ABB RobotStudio station: OpenRobotica_versão15_04_SEM_LETRAS_MASFUNC.rspag

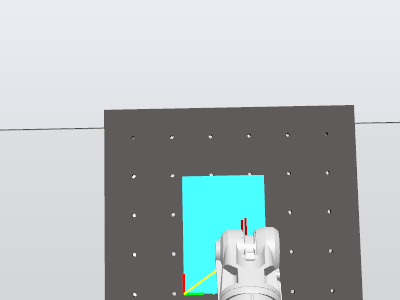
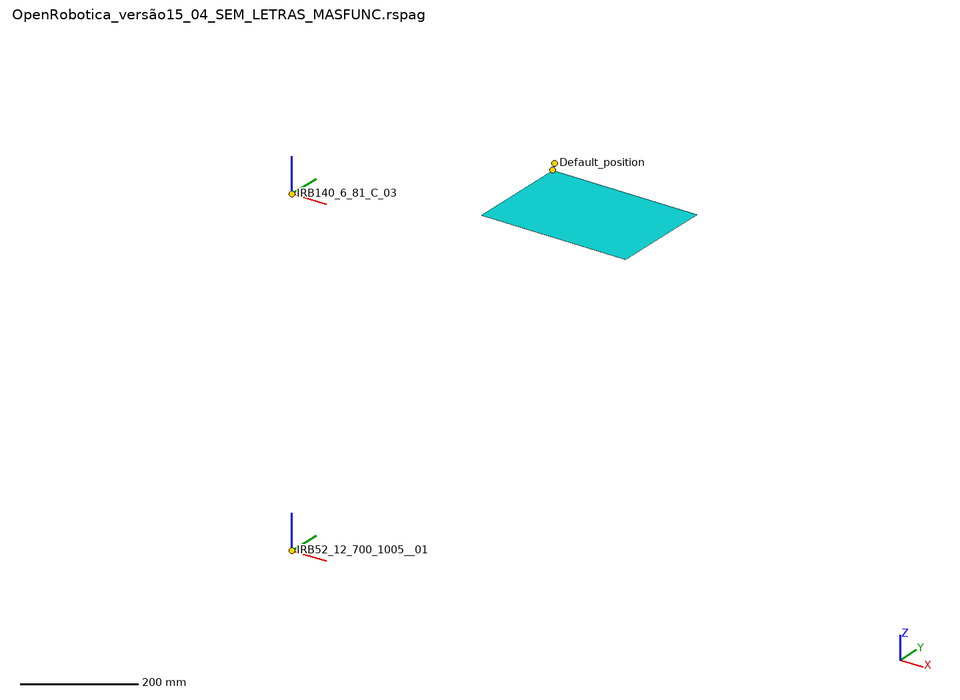
[picture v1: parts stored in the station drawn from their meshes, with robot base, taught points and paths (robot models come from the ABB library and are not in the file)]
--- station ---
Station V1 (saved by RobotStudio 24.1.10693.0)
Controller Robot_ISEP_IRB140, task T_ROB1: task frame (RAPID world) sits at (0, 0, 670) mm in the station
Controller Robot_ISEP_IRB140
  mechanical unit ROB_1: IRB140_6_81_C_03, 6 joints, base frame (0, 0, 0) mm
Controller Robo_open_v2
  mechanical unit ROB_1: IRB52_12_700_1005__01, 6 joints, base frame (0, 0, 0) mm, rotated rx 0 ry 0 rz 90 deg
Layout (positions relative to the parent item):
  - IRB140_6_81_C_03 [mechanism, from %ABB.RobotStudio.Models.IRB140%\IRB140_6_81_C_G_03.rslib] at (0, 0, 670) mm; joint values [-0.036, 0.5458, 0.1215, 0, 0.9034, 3.1056] (rad or m)
  - rob-table [part, from Libraries\rob-table.rslib]
  - pen [mechanism, from Libraries\pen.rslib] at (555, -20, 1029.5) mm, rotated rx 180 ry 0 rz 0 deg
  - paper [part, from Libraries\paper.rslib]
  - IRB52_12_700_1005__01 [mechanism, from %ABB.RobotStudio.Models.IRB52%\IRB52_12_700_1005_G_01.rslib] at (0, 0, 0) mm, rotated rx 0 ry 0 rz 90 deg; joint values [0, 0, 0, 0, 0, 0] (rad or m)
  - A3_Vertical [part] at (450, 125, 790) mm, rotated rx 0 ry 0 rz -90 deg, size 297 x 420 x 0.5 mm
  - A3_Horizontal [part] at (747, 125, 790) mm, rotated rx 0 ry 0 rz 180 deg, size 297 x 420 x 0.5 mm
  - A4_Vertical [part] at (450, 125, 790) mm, rotated rx 0 ry 0 rz -90 deg, size 210 x 297 x 0.5 mm
  - A4_Horizontal [part] at (450, -172, 790) mm, size 210 x 297 x 0.5 mm
  - A5_Vertical [part] at (450, 125, 790) mm, rotated rx 0 ry 0 rz -90 deg, size 148 x 210 x 0.5 mm
  - A5_Horizontal [part] at (450, -85, 790) mm, size 148 x 210 x 0.5 mm
Attachment: pen is attached to IRB140_6_81_C_03 / Link6
Targets, tools, work objects and paths stored in the station and not in the controller backup, written as RAPID:
! task T_ROB1
MODULE Module1
  CONST robtarget Target_Start:=[[0,0,0],[1,0,0,0],[0,0,0,0],[9E+09,9E+09,9E+09,9E+09,9E+09,9E+09]];
ENDMODULE

! task T_ROB1
MODULE DryLetter
  VAR robtarget up_inf_esq1:=[[0,0,0],[1,0,0,0],[0,0,0,0],[9E+09,9E+09,9E+09,9E+09,9E+09,9E+09]];
  VAR robtarget inf_esq1:=[[0,0,0],[1,0,0,0],[0,0,0,0],[9E+09,9E+09,9E+09,9E+09,9E+09,9E+09]];
  VAR robtarget sup_esq:=[[0,0,0],[1,0,0,0],[0,0,0,0],[9E+09,9E+09,9E+09,9E+09,9E+09,9E+09]];
  VAR robtarget sup_dir:=[[0,0,0],[1,0,0,0],[0,0,0,0],[9E+09,9E+09,9E+09,9E+09,9E+09,9E+09]];
  VAR robtarget inf_dir2:=[[0,0,0],[1,0,0,0],[0,0,0,0],[9E+09,9E+09,9E+09,9E+09,9E+09,9E+09]];
  VAR robtarget up_inf_dir2:=[[0,0,0],[1,0,0,0],[0,0,0,0],[9E+09,9E+09,9E+09,9E+09,9E+09,9E+09]];
  VAR robtarget meio_dir:=[[0,0,0],[1,0,0,0],[0,0,0,0],[9E+09,9E+09,9E+09,9E+09,9E+09,9E+09]];
  VAR robtarget meio_esq:=[[0,0,0],[1,0,0,0],[0,0,0,0],[9E+09,9E+09,9E+09,9E+09,9E+09,9E+09]];
  VAR robtarget up_final:=[[0,0,0],[1,0,0,0],[0,0,0,0],[9E+09,9E+09,9E+09,9E+09,9E+09,9E+09]];
  VAR robtarget sup_centro:=[[0,0,0],[1,0,0,0],[0,0,0,0],[9E+09,9E+09,9E+09,9E+09,9E+09,9E+09]];
  VAR robtarget meio_centro:=[[0,0,0],[1,0,0,0],[0,0,0,0],[9E+09,9E+09,9E+09,9E+09,9E+09,9E+09]];
  VAR robtarget inf_centro:=[[0,0,0],[1,0,0,0],[0,0,0,0],[9E+09,9E+09,9E+09,9E+09,9E+09,9E+09]];
  VAR robtarget up_meio_esq:=[[0,0,0],[1,0,0,0],[0,0,0,0],[9E+09,9E+09,9E+09,9E+09,9E+09,9E+09]];
  VAR robtarget sup_dir_meio:=[[0,0,0],[1,0,0,0],[0,0,0,0],[9E+09,9E+09,9E+09,9E+09,9E+09,9E+09]];
  VAR robtarget inf_dir_meio:=[[0,0,0],[1,0,0,0],[0,0,0,0],[9E+09,9E+09,9E+09,9E+09,9E+09,9E+09]];
  PROC Letra_A()
    MoveJ up_inf_esq1,v100,fine,pen\WObj:=Workobject_Paper;
    MoveL inf_esq1,v100,fine,pen\WObj:=Workobject_Paper;
    MoveL sup_esq,v100,z0,pen\WObj:=Workobject_Paper;
    MoveL sup_dir,v100,z0,pen\WObj:=Workobject_Paper;
    MoveL inf_dir2,v100,fine,pen\WObj:=Workobject_Paper;
    MoveL up_inf_dir2,v100,z0,pen\WObj:=Workobject_Paper;
    MoveL meio_dir,v100,z0,pen\WObj:=Workobject_Paper;
    MoveL meio_esq,v100,fine,pen\WObj:=Workobject_Paper;
    MoveL up_final,v100,z0,pen\WObj:=Workobject_Paper;
  ENDPROC
  PROC Letra_B()
    MoveJ target_oInf1Esq1,v100,fine,pen\WObj:=Workobject_Paper;
    MoveL target_oInf1Esq1,v100,fine,pen\WObj:=Workobject_Paper;
    MoveL target_oInf1Esq1,v100,fine,pen\WObj:=Workobject_Paper;
  ENDPROC
  PROC Letra_F()
    MoveJ up_inf_esq1,v100,fine,pen\WObj:=Workobject_Paper;
  ENDPROC
  PROC Space_letter()
    MoveJ target_oInf1Esq1,v100,fine,pen\WObj:=Workobject_Paper;
  ENDPROC
ENDMODULE

! task T_ROB1
MODULE Math
  PROC impressmenu()
    write_string;
    calculo_size;
    settingsTextMenu;
    settingsPageMenu;
    write_string;
    impress_mecanism;
  ENDPROC
ENDMODULE

! task T_ROB1
MODULE Menu
  PROC start_default()
    WaitTime 3;
  ENDPROC
  PROC principal_menu()
    menu_text;
    menu_paper;
    impressmenu;
  ENDPROC
ENDMODULE

! task T_ROB1
MODULE Print
  PROC impress_mecanism()
    draw;
    MoveJ Default_position,v1000,fine,pen\WObj:=Workobject_Paper;
    WaitTime 5;
  ENDPROC
ENDMODULE

! task T_ROB1
MODULE Fonts
  VAR robtarget target_oInf2Centro:=[[0,0,0],[1,0,0,0],[0,0,0,0],[9E+09,9E+09,9E+09,9E+09,9E+09,9E+09]];
  VAR robtarget target_oInf2Esq2:=[[0,0,0],[1,0,0,0],[0,0,0,0],[9E+09,9E+09,9E+09,9E+09,9E+09,9E+09]];
  VAR robtarget target_oInf2Dir1:=[[0,0,0],[1,0,0,0],[0,0,0,0],[9E+09,9E+09,9E+09,9E+09,9E+09,9E+09]];
  VAR robtarget target_oCentroDir1:=[[0,0,0],[1,0,0,0],[0,0,0,0],[9E+09,9E+09,9E+09,9E+09,9E+09,9E+09]];
  VAR robtarget target_oSup1Dir1:=[[0,0,0],[1,0,0,0],[0,0,0,0],[9E+09,9E+09,9E+09,9E+09,9E+09,9E+09]];
  VAR robtarget target_oSup2Esq2:=[[0,0,0],[1,0,0,0],[0,0,0,0],[9E+09,9E+09,9E+09,9E+09,9E+09,9E+09]];
  VAR robtarget target_oSup2Centro:=[[0,0,0],[1,0,0,0],[0,0,0,0],[9E+09,9E+09,9E+09,9E+09,9E+09,9E+09]];
  VAR robtarget target_oSup2Dir1:=[[0,0,0],[1,0,0,0],[0,0,0,0],[9E+09,9E+09,9E+09,9E+09,9E+09,9E+09]];
ENDMODULE


--- Backups/Robot_ISEP_IRB140/RAPID/TASK1/PROGMOD/CalibData.mod ---
MODULE CalibData
    PERS tooldata tWeldGun:=[TRUE,[[125.800591275,0,391.268161315],[0.898794046,0,0.438371147,0]],[3,[0,0,100],[0,1,0,0],0,0,0]];
    PERS tooldata pen:=[TRUE,[[0,0,139],[1,0,0,0]],[0.5,[0,0,20],[1,0,0,0],0,0,0]];
    TASK PERS wobjdata Workobject_Paper:=[FALSE,TRUE,"",[[450,125,118],[0,1,0,0]],[[50,50,0],[1,0,0,0]]];

    CONST robtarget Origem:=[[-50,-50,-2.5],[1,0,0,0],[0,0,0,0],[9E+09,9E+09,9E+09,9E+09,9E+09,9E+09]];
    CONST robtarget Default_position:=[[55,95,-102.5],[1,0,0,0],[0,0,0,0],[9E+09,9E+09,9E+09,9E+09,9E+09,9E+09]];
ENDMODULE

--- Backups/Robot_ISEP_IRB140/RAPID/TASK1/PROGMOD/Fonts.mod ---
MODULE Fonts

    ! Offset Z
    VAR num offsetZ := 10;

    ! On the paper

    VAR robtarget target_oInf1Esq1;
    VAR robtarget target_oInf1Esq2;
    VAR robtarget target_oInf1Centro;
    VAR robtarget target_oInf1Dir1;
    VAR robtarget target_oInf1Dir2;

    VAR robtarget target_oInf2Esq1;
    VAR robtarget target_oInf2Esq2;
    VAR robtarget target_oInf2Centro;
    VAR robtarget target_oInf2Dir1;
    VAR robtarget target_oInf2Dir2;

    VAR robtarget target_oCentroEsq1;
    VAR robtarget target_oCentroEsq2;
    VAR robtarget target_oCentroCentro;
    VAR robtarget target_oCentroDir1;
    VAR robtarget target_oCentroDir2;

    VAR robtarget target_oSup1Esq1;
    VAR robtarget target_oSup1Esq2;
    VAR robtarget target_oSup1Centro;
    VAR robtarget target_oSup1Dir1;
    VAR robtarget target_oSup1Dir2;

    VAR robtarget target_oSup2Esq1;
    VAR robtarget target_oSup2Esq2;
    VAR robtarget target_oSup2Centro;
    VAR robtarget target_oSup2Dir1;
    VAR robtarget target_oSup2Dir2;

    ! Above the paper

    VAR robtarget target_aInf1Esq1;
    VAR robtarget target_aInf1Esq2;
    VAR robtarget target_aInf1Centro;
    VAR robtarget target_aInf1Dir1;
    VAR robtarget target_aInf1Dir2;

    VAR robtarget target_aInf2Esq1;
    VAR robtarget target_aInf2Esq2;
    VAR robtarget target_aInf2Centro;
    VAR robtarget target_aInf2Dir1;
    VAR robtarget target_aInf2Dir2;

    VAR robtarget target_aCentroEsq1;
    VAR robtarget target_aCentroEsq2;
    VAR robtarget target_aCentroCentro;
    VAR robtarget target_aCentroDir1;
    VAR robtarget target_aCentroDir2;

    VAR robtarget target_aSup1Esq1;
    VAR robtarget target_aSup1Esq2;
    VAR robtarget target_aSup1Centro;
    VAR robtarget target_aSup1Dir1;
    VAR robtarget target_aSup1Dir2;

    VAR robtarget target_aSup2Esq1;
    VAR robtarget target_aSup2Esq2;
    VAR robtarget target_aSup2Centro;
    VAR robtarget target_aSup2Dir1;
    VAR robtarget target_aSup2Dir2;

    ! Last Position
    VAR robtarget last_position;

PROC draw( )

       TPWrite "Caracter a Imprimir: " + character;

       target_aInf1Esq1 := Offs(origem, coord_y_letter, coord_x_letter, -offsetZ);
       target_oInf1Esq1 := Offs(origem, coord_y_letter, coord_x_letter, 0);
       target_aInf1Dir2 := Offs(target_aInf1Esq1, 0, comprimento_letras,0);
       target_oInf1Dir2 := Offs(target_oInf1Esq1, 0, comprimento_letras,0);

       target_aSup1Esq1 := Offs(target_aInf1Esq1, altura_letras, 0, 0);
       target_oSup1Esq1 := Offs(target_oInf1Esq1, altura_letras, 0, 0);
       target_aSup1Dir2 := Offs(target_aSup1Esq1, 0, comprimento_letras,0);
       target_oSup1Dir2 := Offs(target_oSup1Esq1, 0, comprimento_letras,0);

       IF "Classic" = text_FontType THEN
	        IF "A" = character OR "a" = character THEN
	            ! Instructions to draw letter "A"
                    target_oCentroDir2 := Offs (target_oInf1Dir2, altura_letras/2 , 0, 0);
                    target_oCentroEsq1 := Offs (target_oCentroDir2, 0, -comprimento_letras, 0);
                    target_aCentroEsq1 := Offs (target_oCentroEsq1, 0, 0, -10);

                ! definição Trajeto

                    ! adaptar origem

                    MoveJ target_aInf1Esq1, v100, fine, pen\WObj:=Workobject_Paper;
                    MoveL target_oInf1Esq1, v100, fine, pen\WObj:=Workobject_Paper;
                    MoveL target_oSup1Esq1, v100, z50, pen\WObj:=Workobject_Paper;
                    MoveL target_oSup1Dir2, v100, z50, pen\WObj:=Workobject_Paper;
                    MoveL target_oInf1Dir2, v100, fine, pen\WObj:=Workobject_Paper;
                    MoveL target_oCentroDir2, v100, z0, pen\WObj:=Workobject_Paper;
                    MoveL target_oCentroEsq1, v100, fine, pen\WObj:=Workobject_Paper;
                    MoveL target_aCentroEsq1, v100, fine, pen\WObj:=Workobject_Paper;

                    !last_position := CRobT(\Tool:=pen\WObj:=Workobject_Paper);

	        ELSEIF "B" = character OR "b" = character THEN
	            ! Instructions to draw letter "B"
                target_oSup1Centro := Offs (target_oSup1Esq1, 0, comprimento_letras/2, 0);
                target_oSup2Dir2 := Offs (target_oSup1Centro, -altura_letras/4, comprimento_letras/2,0);
                target_oCentroCentro := Offs (target_oSup1Centro, -altura_letras/2, 0, 0); ! no MoveL tenho de fazer z30 (experimentar -> se quiser curva maior, fazer valor > 30)
                target_oInf2Dir2 := Offs (target_oCentroCentro, -altura_letras/4, comprimento_letras/2,0);
                target_oCentroEsq1 := Offs(target_oCentroCentro,0,-comprimento_letras/2, 0);
                target_oInf1Centro := Offs (target_oCentroCentro, -altura_letras/2, 0, 0); !z30

                ! definição Trajeto

                MoveJ target_oInf1Esq1, v100, fine, pen\WObj:=Workobject_Paper;
                MoveL target_oInf1Esq1, v100, fine, pen\WObj:=Workobject_Paper;
                MoveL target_oSup1Esq1, v100, fine, pen\WObj:=Workobject_Paper;
                MoveL target_oSup1Centro, v100, z0, pen\WObj:=Workobject_Paper;
                MoveC target_oSup2Dir2, target_oCentroCentro, v100, fine, pen\WObj:=Workobject_Paper;
                MoveL target_oCentroEsq1, v100, fine, pen\WObj:=Workobject_Paper;
                MoveL target_oCentroCentro, v100, fine, pen\WObj:=Workobject_Paper;
                MoveC target_oInf2Dir2 ,target_oInf1Centro, v100, fine, pen\WObj:=Workobject_Paper;
                MoveL target_oInf1Esq1, v100, fine, pen\WObj:=Workobject_Paper;

                MoveL target_aInf1Esq1, v100, z0, pen\WObj:=Workobject_Paper;

                last_position := CRobT(\Tool:=pen\WObj:=Workobject_Paper);

	        ELSEIF "C" = character OR "c" = character THEN
	            ! Instructions to draw letter "C"
                !Don't Finish

                target_oSup2Dir2 := Offs(target_oSup1Dir2,-altura_letras/4,0,0);
                target_aSup2Dir2 := Offs(target_oSup2Dir2,0,0, - offsetZ);
                target_oSup1Centro := Offs(target_oSup1Esq1,0,comprimento_letras/2,0);
                target_oSup2Esq1 := Offs(target_oSup1Esq1,-altura_letras/4,0,0);
                target_oInf2Esq1 := Offs(target_oInf1Esq1,altura_letras/4,0,0);
                target_oInf1Centro := Offs(target_oInf1Esq1,0,comprimento_letras/2,0);
                target_oInf2Dir2 := Offs(target_oInf1Esq1,altura_letras/4,0,0);
                target_aInf2Dir2 := Offs(target_oInf2Dir2,0,0, - offsetZ);


                !traject
                MoveJ target_aSup2Dir2, v100, fine, pen\WObj:=Workobject_Paper;
                MoveL target_oSup2Dir2, v100, fine, pen\WObj:=Workobject_Paper;
                MoveC target_oSup1Centro, target_oSup2Esq1, v100, fine, pen\WObj:=Workobject_Paper;
                MoveL target_oInf2Esq1, v100, fine, pen\WObj:=Workobject_Paper;
                MoveC target_oInf1Centro, target_oInf2Dir2, v100, fine, pen\WObj:=Workobject_Paper;
                MoveL target_aInf2Dir2, v100, fine, pen\WObj:=Workobject_Paper;

	        ELSEIF "D" = character OR "d" = character THEN
	            ! Instructions to draw letter "D"
	        ELSEIF "E" = character OR "e" = character THEN
	            ! Instructions to draw letter "E"
	        ELSEIF "F" = character OR "f" = character THEN
	            ! Instructions to draw letter "F"
	        ELSEIF "G" = character OR "g" = character THEN
	            ! Instructions to draw letter "G"
	        ELSEIF "H" = character OR "h" = character THEN
	            ! Instructions to draw letter "H"
	        ELSEIF "I" = character OR "i" = character THEN
	            ! Instructions to draw letter "I"
	        ELSEIF "J" = character OR "j" = character THEN
	            ! Instructions to draw letter "J"
	        ELSEIF "K" = character OR "k" = character THEN
	            ! Instructions to draw letter "K"
	        ELSEIF "L" = character OR "l" = character THEN
	            ! Instructions to draw letter "L"
	       ELSEIF "M" = character OR "m" = character THEN
	            ! Instructions to draw letter "M"
                target_aCentroCentro := Offs( target_aInf1Esq1 , altura_letras/2 , comprimento_letras/2 , 0);
                target_oCentroCentro := Offs( target_oInf1Esq1 , altura_letras/2 , comprimento_letras/2 , 0);

		        ! Movement
		        MoveJ target_aInf1Esq1, v100, fine, pen\WObj:=Workobject_Paper;
		        MoveL target_oInf1Esq1, v100, fine, pen\WObj:=Workobject_Paper;
		        MoveL target_oSup1Esq1, v100, fine, pen\WObj:=Workobject_Paper;
		        MoveL target_oCentroCentro, v100, fine, pen\WObj:=Workobject_Paper;
		        MoveL target_oSup1Dir2, v100, fine, pen\WObj:=Workobject_Paper;
		        MoveL target_oInf1Dir2, v100, fine, pen\WObj:=Workobject_Paper;
		        MoveL target_aInf1Dir2, v100, fine, pen\WObj:=Workobject_Paper;

	        ELSEIF "N" = character OR "n" = character THEN
		        ! Movement
		        MoveJ target_aInf1Esq1, v100, fine, pen\WObj:=Workobject_Paper;
		        MoveL target_oInf1Esq1, v100, fine, pen\WObj:=Workobject_Paper;
		        MoveL target_oSup1Esq1, v100, fine, pen\WObj:=Workobject_Paper;
		        MoveL target_oInf1Dir2, v100, fine, pen\WObj:=Workobject_Paper;
		        MoveL target_oSup1Dir2, v100, fine, pen\WObj:=Workobject_Paper;
		        MoveL target_aSup1Dir2, v100, fine, pen\WObj:=Workobject_Paper;

	        ELSEIF "O" = character OR "o" = character THEN
	            ! Instructions to draw letter "O"
                target_aSup1Centro := Offs( target_aInf1Esq1 , altura_letras , comprimento_letras/2 , 0);
                target_oSup1Centro := Offs( target_oInf1Esq1 , altura_letras , comprimento_letras/2 , 0);

                target_aInf1Centro := Offs( target_aInf1Esq1 , 0 , comprimento_letras/2 , 0);
                target_oInf1Centro := Offs( target_oInf1Esq1 , 0 , comprimento_letras/2 , 0);

                target_aCentroDir2 := Offs( target_aInf1Esq1 , altura_letras/2 , comprimento_letras , 0);
                target_oCentroDir2 := Offs( target_oInf1Esq1 , altura_letras/2 , comprimento_letras , 0);

                target_aCentroEsq1 := Offs( target_aInf1Esq1 , altura_letras/2 , 0 , 0);
                target_oCentroEsq1 := Offs( target_oInf1Esq1 , altura_letras/2 , 0 , 0);


		        ! Movement
		        MoveJ target_aCentroEsq1, v100, fine, pen\WObj:=Workobject_Paper;
		        MoveL target_oCentroEsq1, v100, fine, pen\WObj:=Workobject_Paper;
		        MoveC target_oSup1Centro , target_oCentroDir2 , v100, fine, pen\WObj:=Workobject_Paper;
		        MoveC target_oInf1Centro , target_oCentroEsq1 , v100, fine, pen\WObj:=Workobject_Paper;
		        MoveL target_aCentroEsq1, v100, fine, pen\WObj:=Workobject_Paper;

	        ELSEIF "P" = character OR "p" = character THEN
	            ! Instructions to draw letter "P"
                target_aSup2Dir2 := Offs( target_aInf1Esq1 , altura_letras*3/4 , comprimento_letras, 0);
                target_oSup2Dir2 := Offs( target_oInf1Esq1 , altura_letras*3/4 , comprimento_letras, 0);

                target_aCentroEsq1 := Offs( target_aInf1Esq1 , altura_letras/2 , 0, 0);
                target_oCentroEsq1 := Offs( target_oInf1Esq1 , altura_letras/2 , 0, 0);

                target_aCentroEsq2 := Offs( target_aInf1Esq1 , altura_letras/2 , comprimento_letras *1/4, 0);
                target_oCentroEsq2 := Offs( target_oInf1Esq1 , altura_letras/2 , comprimento_letras *1/4, 0);

                target_aSup1Esq2 := Offs( target_aInf1Esq1 , altura_letras , comprimento_letras *1/4, 0);
                target_oSup1Esq2 := Offs( target_oInf1Esq1 , altura_letras , comprimento_letras *1/4, 0);

		        ! Movement
		        MoveJ target_aInf1Esq1, v100, fine, pen\WObj:=Workobject_Paper;
		        MoveL target_oInf1Esq1, v100, fine, pen\WObj:=Workobject_Paper;
		        MoveL target_oSup1Esq1, v100, fine, pen\WObj:=Workobject_Paper;
		        MoveL target_oSup1Esq2, v100, fine, pen\WObj:=Workobject_Paper;
		        MoveC target_oSup2Dir2 , target_oCentroEsq2 , v100, fine, pen\WObj:=Workobject_Paper;
		        MoveL target_oCentroEsq1, v100, fine, pen\WObj:=Workobject_Paper;
		        MoveL target_aCentroEsq1, v100, fine, pen\WObj:=Workobject_Paper;


	        ELSEIF "Q" = character OR "q" = character THEN
	            ! Instructions to draw letter "Q"
	        ELSEIF "R" = character OR "r" = character THEN
	            ! Instructions to draw letter "R"
	        ELSEIF "S" = character OR "s" = character THEN
	            ! Instructions to draw letter "S"
                target_aSup2Dir2 := Offs( target_aInf1Esq1 , altura_letras * 3/4 , comprimento_letras , 0);
                target_oSup2Dir2 := Offs( target_oInf1Esq1 , altura_letras * 3/4 , comprimento_letras , 0);


                target_aInf2Esq1 := Offs( target_aInf1Esq1 , altura_letras * 1/4 , 0 , 0);
                target_oInf2Esq1 := Offs( target_oInf1Esq1 , altura_letras * 1/4 , 0 , 0);

                target_aInf1Centro := Offs( target_aInf1Esq1 , 0 , comprimento_letras/2 , 0);
                target_oInf1Centro := Offs( target_oInf1Esq1 , 0 , comprimento_letras/2 , 0);
                target_aSup1Centro := Offs( target_aInf1Esq1 , altura_letras , comprimento_letras/2 , 0);
                target_oSup1Centro := Offs( target_oInf1Esq1 , altura_letras , comprimento_letras/2 , 0);

                target_aInf2Dir2 := Offs( target_aInf1Esq1 , altura_letras * 1/4 , comprimento_letras , 0);
                target_oInf2Dir2 := Offs( target_oInf1Esq1 , altura_letras * 1/4 , comprimento_letras , 0);

                target_aCentroCentro := Offs( target_aInf1Esq1 , altura_letras/2 , comprimento_letras/2 , 0);
                target_oCentroCentro := Offs( target_oInf1Esq1 , altura_letras/2 , comprimento_letras/2 , 0);

                target_aSup2Esq1 := Offs( target_aInf1Esq1 , altura_letras * 3/4 , 0 , 0);
                target_oSup2Esq1 := Offs( target_oInf1Esq1 , altura_letras * 3/4 , 0 , 0);

                target_oCentroEsq1 := Offs( target_oInf1Esq1, altura_letras / 2 ,0,0);

                target_oCentroDir2 := Offs ( target_oInf1Dir2, altura_letras / 2 , 0 , 0);
		        ! Movement
		        MoveJ target_aSup2Dir2, v100, fine, pen\WObj:=Workobject_Paper;
		        MoveL target_oSup2Dir2, v100, fine, pen\WObj:=Workobject_Paper;
		        MoveC target_oSup1Centro , target_oSup2Esq1 , v100, fine, pen\WObj:=Workobject_Paper;

                MoveL target_oCentroEsq1, v100, z150, pen\WObj:=Workobject_Paper;
                MoveL target_oCentroCentro, v100, fine, pen\WObj:=Workobject_Paper;
                MoveL target_oCentroDir2, v100, z150, pen\WObj:=Workobject_Paper;
                MoveL target_oInf2Dir2, v100, fine, pen\WObj:=Workobject_Paper;

                MoveC target_oInf1Centro , target_oInf2Esq1 , v100, fine, pen\WObj:=Workobject_Paper;
		        MoveL target_aInf2Esq1, v100, fine, pen\WObj:=Workobject_Paper;


	        ELSEIF "T" = character OR "t" = character THEN
	            ! Instructions to draw letter "T"
                target_aInf1Centro := Offs( target_aInf1Esq1 , 0 , comprimento_letras/2 , 0);
                target_oInf1Centro := Offs( target_oInf1Esq1 , 0 , comprimento_letras/2 , 0);
                target_aSup1Centro := Offs( target_aInf1Esq1 , altura_letras , comprimento_letras/2 , 0);
                target_oSup1Centro := Offs( target_oInf1Esq1 , altura_letras , comprimento_letras/2 , 0);

		        ! Movement
		        MoveJ target_aSup1Esq1, v100, fine, pen\WObj:=Workobject_Paper;
		        MoveL target_oSup1Esq1, v100, fine, pen\WObj:=Workobject_Paper;
		        MoveL target_oSup1Dir2, v100, fine, pen\WObj:=Workobject_Paper;
		        MoveL target_oSup1Centro, v100, fine, pen\WObj:=Workobject_Paper;
		        MoveL target_oInf1Centro, v100, fine, pen\WObj:=Workobject_Paper;
		        MoveL target_aInf1Centro, v100, fine, pen\WObj:=Workobject_Paper;

	        ELSEIF "U" = character OR "u" = character THEN
	            ! Instructions to draw letter "U"
                target_aInf1Centro := Offs( target_aInf1Esq1 , 0 , comprimento_letras/2 , 0);
                target_oInf1Centro := Offs( target_oInf1Esq1 , 0 , comprimento_letras/2 , 0);
                target_aInf2Esq1 := Offs( target_aInf1Esq1 , altura_letras/4 , 0 , 0);
                target_oInf2Esq1 := Offs( target_oInf1Esq1 , altura_letras/4 , 0 , 0);
                target_aInf2Dir2 := Offs( target_aInf1Esq1 , altura_letras/4 , comprimento_letras , 0);
                target_oInf2Dir2 := Offs( target_oInf1Esq1 , altura_letras/4 , comprimento_letras , 0);

		        ! Movement
		        MoveJ target_aSup1Esq1, v100, fine, pen\WObj:=Workobject_Paper;
		        MoveL target_oSup1Esq1, v100, fine, pen\WObj:=Workobject_Paper;
		        MoveL target_oInf2Esq1, v100, fine, pen\WObj:=Workobject_Paper;
		        MoveC target_oInf1Centro , target_oInf2Dir2 , v100, fine, pen\WObj:=Workobject_Paper;
		        MoveL target_oSup1Dir2, v100, fine, pen\WObj:=Workobject_Paper;
		        MoveL target_aSup1Dir2, v100, fine, pen\WObj:=Workobject_Paper;


	        ELSEIF "V" = character OR "v" = character THEN
	            ! Instructions to draw letter "V"
                target_aInf1Centro := Offs( target_aInf1Esq1 , 0 , comprimento_letras/2 , 0);
                target_oInf1Centro := Offs( target_oInf1Esq1 , 0 , comprimento_letras/2 , 0);

		        ! Movement
		        MoveJ target_aSup1Esq1, v100, fine, pen\WObj:=Workobject_Paper;
		        MoveL target_oSup1Esq1, v100, fine, pen\WObj:=Workobject_Paper;
		        MoveL target_oInf1Centro, v100, fine, pen\WObj:=Workobject_Paper;
		        MoveL target_oSup1Dir2, v100, fine, pen\WObj:=Workobject_Paper;
		        MoveL target_aSup1Dir2, v100, fine, pen\WObj:=Workobject_Paper;
		        !MoveL target_aInf1Dir2, v100, fine, pen\WObj:=Workobject_Paper;

	        ELSEIF "W" = character OR "w" = character THEN
	            ! Instructions to draw letter "W"
                target_aCentroCentro := Offs( target_aInf1Esq1 , altura_letras/2 , comprimento_letras/2 , 0);
                target_oCentroCentro := Offs( target_oInf1Esq1 , altura_letras/2 , comprimento_letras/2 , 0);
                target_aInf1Esq2 := Offs( target_aInf1Esq1 , 0 , comprimento_letras/4 , 0);
                target_oInf1Esq2 := Offs( target_oInf1Esq1 , 0 , comprimento_letras/4 , 0);
                target_aInf1Dir1 := Offs( target_aInf1Esq1 , 0 , comprimento_letras*3/4 , 0);
                target_oInf1Dir1 := Offs( target_oInf1Esq1 , 0 , comprimento_letras*3/4 , 0);

		        ! Movement
		        MoveJ target_aSup1Esq1, v100, fine, pen\WObj:=Workobject_Paper;
		        MoveL target_oSup1Esq1, v100, fine, pen\WObj:=Workobject_Paper;
		        MoveL target_oInf1Esq2, v100, fine, pen\WObj:=Workobject_Paper;
		        MoveL target_oCentroCentro, v100, fine, pen\WObj:=Workobject_Paper;
		        MoveL target_oInf1Dir1, v100, fine, pen\WObj:=Workobject_Paper;
		        MoveL target_oSup1Dir2, v100, fine, pen\WObj:=Workobject_Paper;
		        MoveL target_aSup1Dir2, v100, fine, pen\WObj:=Workobject_Paper;
		        !MoveL target_aInf1Dir2, v100, fine, pen\WObj:=Workobject_Paper;

	        ELSEIF "X" = character OR "x" = character THEN
	            ! Instructions to draw letter "X"

		        ! Movement
		        MoveJ target_aSup1Esq1, v100, fine, pen\WObj:=Workobject_Paper;
		        MoveL target_oSup1Esq1, v100, fine, pen\WObj:=Workobject_Paper;
		        MoveL target_oInf1Dir2, v100, fine, pen\WObj:=Workobject_Paper;
		        MoveL target_aInf1Dir2, v100, fine, pen\WObj:=Workobject_Paper;
		        MoveL target_aSup1Dir2, v100, fine, pen\WObj:=Workobject_Paper;
		        MoveL target_oSup1Dir2, v100, fine, pen\WObj:=Workobject_Paper;
		        MoveL target_oInf1Esq1, v100, fine, pen\WObj:=Workobject_Paper;
		        MoveL target_aInf1Esq1, v100, fine, pen\WObj:=Workobject_Paper;
		        !MoveL target_aInf1Dir2, v100, fine, pen\WObj:=Workobject_Paper;

	        ELSEIF "Y" = character OR "y" = character THEN

	            ! Instructions to draw letter "Y"
                target_aCentroCentro := Offs( target_aInf1Esq1 , altura_letras/2 , comprimento_letras/2 , 0);
                target_oCentroCentro := Offs( target_oInf1Esq1 , altura_letras/2 , comprimento_letras/2 , 0);
                target_aInf1Centro := Offs( target_aInf1Esq1 , 0 , comprimento_letras/2 , 0);
                target_oInf1Centro := Offs( target_oInf1Esq1 , 0 , comprimento_letras/2 , 0);

		        ! Movement
		        MoveJ target_aSup1Esq1, v100, fine, pen\WObj:=Workobject_Paper;
		        MoveL target_oSup1Esq1, v100, fine, pen\WObj:=Workobject_Paper;
		        MoveL target_oCentroCentro, v100, fine, pen\WObj:=Workobject_Paper;
		        MoveL target_oSup1Dir2, v100, fine, pen\WObj:=Workobject_Paper;
		        MoveL target_aSup1Dir2, v100, fine, pen\WObj:=Workobject_Paper;
		        MoveL target_aCentroCentro, v100, fine, pen\WObj:=Workobject_Paper;
		        MoveL target_oCentroCentro, v100, fine, pen\WObj:=Workobject_Paper;
		        MoveL target_oInf1Centro, v100, fine, pen\WObj:=Workobject_Paper;
		        MoveL target_aInf1Centro, v100, fine, pen\WObj:=Workobject_Paper;
		        !MoveL target_aInf1Dir2, v100, fine, pen\WObj:=Workobject_Paper;

	        ELSEIF "Z" = character OR "z" = character THEN
	           ! Instructions to draw letter "Z"

		        ! Movement
		        MoveJ target_aSup1Esq1, v100, fine, pen\WObj:=Workobject_Paper;
		        MoveL target_oSup1Esq1, v100, fine, pen\WObj:=Workobject_Paper;
		        MoveL target_oSup1Dir2, v100, fine, pen\WObj:=Workobject_Paper;
		        MoveL target_oInf1Esq1, v100, fine, pen\WObj:=Workobject_Paper;
		        MoveL target_oInf1Dir2, v100, fine, pen\WObj:=Workobject_Paper;
		        MoveL target_aInf1Dir2, v100, fine, pen\WObj:=Workobject_Paper;

	        ELSEIF " " = character THEN
	            ! Instructions to draw letter " "
                MoveJ target_oInf1Esq1, v100, fine, pen\WObj:=Workobject_Paper;
	        ELSE

	        ENDIF
	      ENDIF
    ENDPROC
ENDMODULE

--- Backups/Robot_ISEP_IRB140/RAPID/TASK1/PROGMOD/MainModule.mod ---
MODULE MainModule

        CONST robtarget Target_10:=[[0,0,0],[1,0,0,0],[0,-1,-2,0],[9E+09,9E+09,9E+09,9E+09,9E+09,9E+09]];
    CONST robtarget Target_20:=[[70,30,0],[1,0,0,0],[0,-1,-2,0],[9E+09,9E+09,9E+09,9E+09,9E+09,9E+09]];
    CONST robtarget Target_30:=[[0,60,0],[1,0,0,0],[0,-1,-2,0],[9E+09,9E+09,9E+09,9E+09,9E+09,9E+09]];
PROC main()
       ! Default sequence to reposition the robot
       startDefault;

       ! Main loop
        WHILE TRUE DO
            mainMenu;
        ENDWHILE


    ENDPROC
    PROC Path_A()
    ENDPROC
ENDMODULE

--- Backups/Robot_ISEP_IRB140/RAPID/TASK1/PROGMOD/Math.mod ---
MODULE Math
    ! ============== Declara??o de Variaveis =======================

    ! Apoio para as perguntas
    VAR num answer_impress;

    ! Write array
    PERS string char_impress;

    VAR num userInputTextLenght := 0;
    VAR num workSpaceWidth;
    VAR num workSpaceLength;
    VAR num letterLenghtAutomated;
    VAR num letterWidthAutomated;
    VAR num text_SpaceLettersAutomated;

    CONST num factorSpaceBetweenLetters := 5;
    CONST num factorHightLetter := 2;

    ! Position text
    VAR num xAvailable := 0 ;
    VAR num yAvailable := 0 ;
    VAR num coord_x_letter;
    VAR num coord_y_letter;

    PROC write_string()
        TPWrite "Insira a(s) palavra(s) pretendida(s) para imprimir.";
        userInputText := UIAlphaEntry(
            \Header:= "Impressão",
            \Message:= ""
            \Icon:=iconInfo
            \InitString:= "OPEN ROBOTICA");
    ENDPROC


    PROC calculateSizeLetterAutomated()
        ! Get the amount of chars in the array of text
        userInputTextLenght := StrLen(userInputText);

        ! Garentee the user actually inserts a text
        IF 0 = userInputTextLenght THEN
              TPWrite "Error : Necessário texto para poder imprimir.";
              errorA := TRUE;
              RETURN ;
        ENDIF

        ! Get the size of the page
        workSpaceWidth := paper_Width - paper_LeftMargin - paper_RightMargin ;
        workSpaceLength := paper_Length - paper_TopMargin - paper_BottomMargin ;

        ! Calculate the width of the text acordingly to fit the page line
        letterWidthAutomated := ( workSpaceWidth - ( ( userInputTextLenght - 1 ) * text_SpaceLetters ) ) DIV userInputTextLenght ;

        FOR I FROM 1 TO 10 DO
            ! Calculate the space required between letters
            text_SpaceLettersAutomated := text_SpaceLetters + letterWidthAutomated DIV factorSpaceBetweenLetters ;

            ! Recalculate the lenght of the text acordingly to fit the page line considering the new spacement
            letterWidthAutomated := ( workSpaceWidth - ( ( userInputTextLenght - 1 ) * text_SpaceLettersAutomated ) ) DIV userInputTextLenght ;
        ENDFOR

        ! Garantee a minimum space between
        IF 0 = text_SpaceLettersAutomated THEN
             text_SpaceLettersAutomated := 0.1;
        ENDIF

        ! Calcule the necessary height of letter
        letterLenghtAutomated := letterWidthAutomated * factorHightLetter;

        IF workSpaceLength  < letterLenghtAutomated  THEN
            letterLenghtAutomated := workSpaceLength ;
        ENDIF
    ENDPROC

    PROC calculateOrigin( )
        IF FALSE = automatic THEN
	        IF "Esquerda" = paper_alignment THEN
	        	xAvailable := paper_LeftMargin;
	        ELSEIF "Direita" = paper_alignment THEN
	        	xAvailable := paper_RightMargin - letterWidthAutomated * userInputTextLenght ;
	        ELSEIF "Centrado" = paper_alignment THEN
	            xAvailable := workSpaceWidth / 2 - letterWidthAutomated * userInputTextLenght ;
	        ELSEIF "Justificado" = paper_alignment THEN
	        	xAvailable := paper_LeftMargin;
	        ENDIF
        ELSEIF TRUE = automatic THEN
	       	xAvailable := paper_LeftMargin;
	        IF 0 = yAvailable THEN
	            yAvailable := paper_Length - paper_TopMargin - letterLenghtAutomated;
	        ELSE
	            yAvailable := coord_y_letter - letterLenghtAutomated - text_SpaceParag ;
	            !Condition to out page
	            IF 0 > yAvailable THEN
                     TPWrite "Error : Fora de página";
                     errorA := TRUE;
                     RETURN;
	            ENDIF
	        ENDIF
        ENDIF

        coord_x_letter := xAvailable;
        coord_y_letter := yAvailable;
    ENDPROC
ENDMODULE

--- Backups/Robot_ISEP_IRB140/RAPID/TASK1/PROGMOD/Menu.mod ---
MODULE Menu

    ! ============== Definition of variables/constants =============================== !

    ! Questions suport
    VAR num answerInitMenu;
    VAR num answerPaperMenu;
    VAR num answerPaperMenu2;
    VAR num answerSettingMenu;
    VAR num answerWriteTextMenu;
    VAR num answerWriteTextMenu2;
    VAR num answerWrittingMenu;
    VAR num answerPrintingMenu;
    VAR num answerDebugMenu;

    ! Variable that stores the text input
    VAR string userInputText ;
    VAR string character;

    ! Dimensions of the format papers (mm)
    CONST num a3Lenght := 297;
    CONST num a3Width := 420;
    CONST num a4Lenght := 210;
    CONST num a4Width := 297;
    CONST num a5Lenght := 148;
    CONST num a5Width := 210;

    ! Initialize the paper characteristics
    VAR string paper_size := "A4";
    VAR string paper_orientation := "Vertical";
    VAR string paper_alignment := "Esquerda";
    VAR num paper_TopMargin := 20;
    VAR num paper_BottomMargin := 20;
    VAR num paper_LeftMargin := 10;
    VAR num paper_RightMargin := 10;
    VAR num paper_Width := a4Lenght;
    VAR num paper_Length := a4Width;

    ! Initialize the text characteristics
    VAR string text_FontType := "Classic";
    VAR num text_SizePT := 12;
    VAR string text_Color := "Black";
    VAR num text_Rotation := 0;
    VAR num text_SpaceLetters := 2;
    VAR num text_SpaceParag := 5;

    ! Initialize letters characteristics
    VAR num letter_lenght := 5;
    VAR num letter_width := 10;

    VAR num paragraph_write := 0;

    VAR bool automatic := FALSE;

    VAR num altura_letras;
    VAR num comprimento_letras;

    VAR bool errorA := FALSE;

    ! ==================== Code - default ========================= !

    ! Process for the inicialization program
    PROC startDefault( )
        ! Clear console
        TPErase;

        MoveJ Default_position,v1000,fine,pen\WObj:=Workobject_Paper;

        ! JumpHome; !TODO
        TPWrite "O robot está pronto a ser operado.";

        WaitTime(1);
    ENDPROC

    ! ==================== Code - mainMenu ======================== !

    PROC mainMenu()
        !Clear console
        TPErase;

        ! Welcome page.
        TPWrite "Plotter & Open Robótica";

        ! Options of the menu
        TPReadFK answerInitMenu ,
                 stEmpty ,
                 "Escrever Manualmente" ,
                 "Definições texto" ,
                 "Definições folha" ,
                 "Imprimir",
                 "Debug";

        IF 1 = answerInitMenu THEN
            writeTextMenu;
        ELSEIF 2 = answerInitMenu THEN
           answersettingMenu := 0;
           settingsTextMenu ;
        ELSEIF 3 = answerInitMenu THEN
            settingsPageMenu ;
        ELSEIF 4 = answerInitMenu THEN
            printingPageMenu ;
        ELSEIF 5 = answerInitMenu THEN
            debugMenu ;
        ENDIF
    ENDPROC

    ! ==================== Code - writeMenu ======================= !

    PROC writeTextMenu( )
        WHILE answerWrittingMenu <> 5 DO
            ! Clear the console
            TPErase;

            TPWrite("Frase a escrever:");
            ! Options to change settings of the page
            TPReadFK answerSettingMenu,
                     userInputText ,
                     "Escrever",
                     stEmpty,
                     stEmpty,
                     stEmpty,
                     "Voltar";

            IF 1 = answersettingMenu THEN
                write_string;

            ELSEIF 2 = answersettingMenu THEN

            ELSEIF 3 = answersettingMenu THEN

            ELSEIF 4 = answersettingMenu THEN

            ELSEIF 5 = answersettingMenu THEN
                answerWrittingMenu := 5;
                ! Back to menu
            ENDIF
        ENDWHILE
        answerWrittingMenu := 0;
    ENDPROC

    ! ==================== Code - settingsText ==================== !

    PROC settingsTextMenu( )
        WHILE answersettingMenu <> 5 DO
            ! Clear the console
            TPErase;

            tpWriteReportSettingsTextMenu;

            ! Options to change settings of the page
            TPReadFK answerSettingMenu,
                     stEmpty ,
                     "Fonte",
                     "Tamanho (pt)",
                     "Cor",
                     "Página seguinte",
                     "Voltar";

            IF 1 = answersettingMenu THEN
                fontTypePageMenu ;

            ELSEIF 2 = answersettingMenu THEN
                TPReadNum text_SizePT, "Qual é o tamanho da letra? (pt) (default = 12)";
                !TODO convert pt to mm

            ELSEIF 3 = answersettingMenu THEN
                fontColorPageMenu ;

            ELSEIF 4 = answersettingMenu THEN
                answersettingMenu := 0;
                settingsTextMenu2 ;

            ELSEIF 5 = answersettingMenu THEN
                answersettingMenu := 5;
                ! Back to menu
            ENDIF

        ENDWHILE
    ENDPROC

    PROC settingsTextMenu2( )
        WHILE answersettingMenu <> 5 DO
            ! Clear the console
            TPErase;

            tpWriteReportSettingsTextMenu;

            ! Options to change settings of the page
            TPReadFK answerSettingMenu,
                     stEmpty ,
                     "Rotação",
                     "Espaçamento entre letras",
                     "Espaçamento entre paragráfos",
                     "Página seguinte",
                     "Voltar";

            IF 1 = answersettingMenu THEN
                TPReadNum text_Rotation, "Qual é a rotação pretendida? (graus)";

            ELSEIF 2 = answersettingMenu THEN
                TPReadNum text_SpaceLetters, "Qual é o espaçamento entre letras? (mm) (default = 2)";

            ELSEIF 3 = answersettingMenu THEN
                TPReadNum text_SpaceParag, "Qual é o espaçamento entre paragráfos? (mm) (default = 5)";

            ELSEIF 4 = answersettingMenu THEN
                answersettingMenu := 0;
                settingsTextMenu3 ;

            ELSEIF 5 = answersettingMenu THEN
                answersettingMenu := 5;
                ! Back to menu
            ENDIF
        ENDWHILE
    ENDPROC

    PROC settingsTextMenu3( )
        WHILE answersettingMenu <> 5 DO
            ! Clear the console
            TPErase;

            tpWriteReportSettingsTextMenu;

            ! Options to change settings of the page
            TPReadFK answerSettingMenu,
                     stEmpty ,
                     "Negrito",
                     "Itálico",
                     "Sublinhado",
                     "Página seguinte",
                     "Voltar";

            IF 1 = answersettingMenu THEN
                 ! Do nothing yet

            ELSEIF 2 = answersettingMenu THEN
                 ! Do nothing yet

            ELSEIF 3 = answersettingMenu THEN
                 ! Do nothing yet

            ELSEIF 4 = answersettingMenu THEN
                answersettingMenu := 0;
                settingsTextMenu ;
            ELSEIF 5 = answersettingMenu THEN
                answersettingMenu := 5;
                ! Back to menu
            ENDIF
        ENDWHILE
    ENDPROC


    PROC tpWriteReportSettingsTextMenu()
        ! Clear the console
        TPErase;

        TPWrite("Definições de Texto:");

        ! Display font type
        TPWrite("Fonte de Letra: " + text_FontType );

        ! Display letter size
        TPWrite "Tamanho de letra:" + NumToStr(text_SizePT,0) + "pt" + "(" + NumToStr(letter_lenght,0) + " mm , " +  NumToStr(letter_width,0) + " mm )";

        ! Display letter color
        TPWrite "Cor de Letra: " + text_Color;

        ! Display letter rotation
        TPWrite "Rotação do texto: " + NumToStr( text_Rotation, 0 ) + " graus";

        ! Display space between letters
        TPWrite "Espaçamento entre letras: " + NumToStr( text_SpaceLetters, 0 ) + " mm";

        ! Display space between paragraphs
        TPWrite "Espaçamento entre parágrafos: " + NumToStr( text_SpaceParag, 0 ) + " mm";
    ENDPROC

    PROC fontTypePageMenu( )
        ! Clear the console
        TPErase;

        tpWriteReportSettingsTextMenu;

        ! Options to change format
        TPReadFK answerWriteTextMenu2,
                 stEmpty ,
                 "Classic" ,
                 "Digital" ,
                 "Fancy" ,
                 stEmpty ,
                 "Voltar" ;

        IF 1 = answerWriteTextMenu2 THEN
            text_FontType := "Classic";

        ELSEIF 2 = answerWriteTextMenu2 THEN
            text_FontType := "Digital";

        ELSEIF 3 = answerWriteTextMenu2 THEN
            text_FontType := "Fancy";

        ELSEIF 4 = answerWriteTextMenu2 THEN
            ! nothing for now (fuction enable)

        ELSEIF 5 = answerWriteTextMenu2 THEN
            answerWriteTextMenu2 := 0 ;
        ENDIF
    ENDPROC

    PROC fontColorPageMenu( )
        ! Clear the console
        TPErase;

        tpWriteReportSettingsTextMenu;

        ! Options to change format
        TPReadFK answerWriteTextMenu2,
                 stEmpty ,
                 "Preto" ,
                 "Azul" ,
                 "Vermelho" ,
                 stEmpty ,
                 "Voltar" ;

        IF 1 = answerWriteTextMenu2 THEN
            text_Color := "Black";

        ELSEIF 2 = answerWriteTextMenu2 THEN
            text_Color := "Blue";

        ELSEIF 3 = answerWriteTextMenu2 THEN
            text_Color := "Red";

        ELSEIF 4 = answerWriteTextMenu2 THEN
            ! nothing for now (fuction enable)

        ELSEIF 5 = answerWriteTextMenu2 THEN
            answerWriteTextMenu2 := 0 ;
        ENDIF
    ENDPROC


    ! ==================== Code - settingsPage ==================== !

    PROC settingsPageMenu( )
        WHILE 5 <> answerPaperMenu DO
            ! Clear the console
            TPErase;

            tpWriteReportSettingsPageMenu;

            ! Options to change settings of the page
            TPReadFK answerPaperMenu,
                     stEmpty ,
                     "Formato",
                     "Orientação",
                     "Margens",
                     "Alinhamento",
                     "Voltar";

            IF 1 = answerPaperMenu THEN
                formatPageMenu ;
                yAvailable := 0;

            ELSEIF 2 = answerPaperMenu THEN
                orientationPageMenu;
                yAvailable := 0;

            ELSEIF 3 = answerPaperMenu THEN
                marginsPageMenu ;

            ELSEIF 4 = answerPaperMenu THEN
                alignmentPageMenu ;

            ELSEIF 5 = answerPaperMenu THEN !Go out in the while
            ENDIF
        ENDWHILE

        answerPaperMenu := 0;
    ENDPROC

    PROC tpWriteReportSettingsPageMenu()
        TPWrite("Definições de p gina:");

        ! Display paper size
        TPWrite "Formato da folha: " + paper_size + " ( " +  NumToStr(paper_Width,0) + " mm, " +  NumToStr(paper_Length,0) + " mm)";

        ! Display paper orientation
        TPWrite "Orientação da folha: " + paper_Orientation;

        ! Display paper margins
        TPWrite "Margens da folha: ";
        TPWrite " " + NumToStr( paper_TopMargin, 0 ) + " (mm) (cabeçalho)," + NumToStr( paper_BottomMargin ,0 ) + " (mm) (rodapé)," ;
        TPWrite " " + NumToStr( paper_LeftMargin, 0 ) + " (mm) (esquerda)," + NumToStr( paper_RightMargin , 0 ) + " (mm) (direita)" ;

        ! Display text alignment
        TPWrite("Alinhamento do texto: " + paper_Alignment );
    ENDPROC

    PROC formatPageMenu( )
        ! Clear the console
        TPErase;

        tpWriteReportSettingsPageMenu;

        ! Options to change format
        TPReadFK answerPaperMenu2,
                 stEmpty ,
                 "A3" ,
                 "A4" ,
                 "A5" ,
                 stEmpty ,
                 "Voltar" ;

        IF 1 = answerPaperMenu2 THEN
            paper_size := "A3" ;

            IF "Vertical" = paper_orientation THEN
                 paper_Width := a3Lenght;
                 paper_Length := a3Width;
            ELSE
                 paper_Width := a3Width;
                 paper_Length := a3Lenght;
            ENDIF

        ELSEIF 2 = answerPaperMenu2 THEN
            paper_size := "A4" ;

            IF "Vertical" = paper_orientation THEN
                 paper_Width := a4Lenght;
                 paper_Length := a4Width;
            ELSE
                 paper_Width := a4Width;
                 paper_Length := a4Lenght;
            ENDIF

        ELSEIF 3 = answerPaperMenu2 THEN
            paper_size := "A5" ;

            IF "Vertical" = paper_orientation THEN
                 paper_Width := a5Lenght;
                 paper_Length := a5Width;
            ELSE
                 paper_Width := a5Width;
                 paper_Length := a5Lenght;
            ENDIF

        ELSEIF 4 = answerPaperMenu2 THEN
            ! nothing for now (fuction enable)

        ELSEIF 5 = answerPaperMenu2 THEN
            answerPaperMenu2 := 0 ;
        ENDIF
    ENDPROC

    PROC orientationPageMenu( )
        ! Clear the console
        TPErase;

        tpWriteReportSettingsPageMenu;

        ! Options to change orientation
        TPReadFK answerPaperMenu2,
                 stEmpty ,
                 "Horizontal" ,
                 "Vertical" ,
                 stEmpty ,
                 stEmpty ,
                 "Voltar" ;

        IF 1 = answerPaperMenu2 THEN
            paper_Orientation := "Horizontal";

        ELSEIF 2 = answerPaperMenu2 THEN
            paper_Orientation := "Vertical";

        ELSEIF 3 = answerPaperMenu2 THEN
            ! nothing for now

        ELSEIF 4 = answerPaperMenu2 THEN
            ! nothing for now

        ELSEIF 5 = answerPaperMenu2 THEN
            answerPaperMenu2 := 0 ;
        ENDIF
    ENDPROC

    PROC marginsPageMenu( )
        ! Clear the console
        TPErase;

        tpWriteReportSettingsPageMenu;

        ! Options to change orientation
        TPReadFK answerPaperMenu2,
                 stEmpty ,
                 "Cabeçalho" ,
                 "Rodapé" ,
                 "Direita" ,
                 "Esquerda" ,
                 "Voltar" ;

        ! TODO does nothing at the moment

        IF 1 = answerPaperMenu2 THEN
            TPReadNum paper_TopMargin, "Qual é o valor da margem do cabe alho? (mm)";

        ELSEIF 2 = answerPaperMenu2 THEN
            TPReadNum paper_BottomMargin, "Qual é o valor da margem do rodap ? (mm)";

        ELSEIF 3 = answerPaperMenu2 THEN
            TPReadNum paper_RightMargin, "Qual é o valor da margem direita? (mm)";

        ELSEIF 4 = answerPaperMenu2 THEN
            TPReadNum paper_LeftMargin, "Qual é o valor da margem esquerda? (mm)";

        ELSEIF 5 = answerPaperMenu2 THEN
            answerPaperMenu2 := 0 ;
        ENDIF
    ENDPROC

    PROC alignmentPageMenu( )
        ! Clear the console
        TPErase;

        tpWriteReportSettingsPageMenu;

        ! Options to change orientation
        TPReadFK answerPaperMenu2,
                 stEmpty ,
                 "Centro" ,
                 "Esquerda" ,
                 "Direita" ,
                 "Justificado" ,
                 "Voltar" ;

        IF 1 = answerPaperMenu2 THEN
            paper_Alignment := "Centro";

        ELSEIF 2 = answerPaperMenu2 THEN
            paper_Alignment := "Esquerda";

        ELSEIF 3 = answerPaperMenu2 THEN
            paper_Alignment := "Direita";

        ELSEIF 4 = answerPaperMenu2 THEN
            paper_Alignment := "Justificado";

        ELSEIF 5 = answerPaperMenu2 THEN
            answerPaperMenu2 := 0 ;
        ENDIF
    ENDPROC


    !===================== Code - ImpressMenu ============================

    PROC printingPageMenu()
         VAR num x := 1;
        WHILE answerPrintingMenu = 4 OR answerPrintingMenu = 0 DO
           ! Clear the console
           TPErase;

           IF 1 = x THEN
                TPWrite "Texto a ser impresso";
                TPWrite userInputText;
    	        x := 2;
            ELSEIF 2 = X THEN
	            tpWriteReportSettingsTextMenu;
    	        x := 3;
            ELSE
                tpWriteReportSettingsPageMenu;
    	        x := 1;
            ENDIF

            ! Options to change settings of the page
            TPReadFK answerPrintingMenu,
                     stEmpty ,
                     "Automático",
                     "Manual",
                     "Ficheiro",
                     "Scroll",
                     "Voltar";

            IF 1 = answerPrintingMenu THEN
                automaticPrinting;

            ELSEIF 2 = answerPrintingMenu THEN
                !manualPriting;
            ELSEIF 3 = answerPrintingMenu THEN
                !filesPriting;
            ELSEIF 4 = answerPrintingMenu THEN

            ELSEIF 5 = answerPrintingMenu THEN
                answerPrintingMenu := 5;
                ! Back to menu
            ENDIF
        ENDWHILE
        answerPrintingMenu := 0;
    ENDPROC


    PROC automaticPrinting()
        automatic := TRUE;
        calculateSizeLetterAutomated;
        calculateOrigin;
        IF TRUE = errorA THEN
            automatic := FALSE;
            errorA := FALSE;
            RETURN;
        ENDIF

        altura_letras := letterLenghtAutomated ;
        comprimento_letras := letterWidthAutomated ;

        impressMecanism;
        automatic := FALSE;
    ENDPROC

    ! ==================== Code - debugMenu ==================== !

    PROC debugMenu( )
        ! Clear the console
        TPErase;

        !TPRead
    ENDPROC
ENDMODULE

--- Backups/Robot_ISEP_IRB140/RAPID/TASK1/PROGMOD/Module1.mod ---
MODULE Module1
    PROC Path_10()
        MoveL Default_position,v1000,z100,pen\WObj:=Workobject_Paper;
        MoveL Origem,v1000,z100,pen\WObj:=Workobject_Paper;
    ENDPROC
ENDMODULE

--- Backups/Robot_ISEP_IRB140/RAPID/TASK1/PROGMOD/Print.mod ---
MODULE Print
    CONST num time := 5;

    PROC impressMecanism()
        TPErase;
        !TPWrite NumtoStr(coord_y_letter,0);
        TPWrite "A imprimir  ...";

		FOR i FROM 1 TO StrLen( userInputText ) DO
            character := StrPart( userInputText, i, 1);
            draw;

            !TPWrite NumToStr(coord_x_letter,0);
            !WaitTime(2);
            !Calculate new point center

            IF TRUE = automatic THEN
                coord_x_letter := coord_x_letter + letterWidthAutomated + text_SpaceLettersAutomated ;
            ELSE
                coord_x_letter := coord_x_letter + letter_width + text_SpaceLetters ;
            ENDIF
		ENDFOR

        TPWrite "Impressão Feita";

        MoveJ Default_position, v100 , fine , pen\WObj:=Workobject_Paper ;
        WaitTime( time );
    ENDPROC
ENDMODULE

--- Backups/Robo_open_v2/RAPID/TASK0/SYSMOD/guisocks.sys ---
module guisocks(sysmodule)

   pers num nGUISockCmdId    := 0;
   pers num nGUISockClientId := 0;
   pers num nGUISockSerNo    := 0;

   pers num nGUISockPars{10}      := [0,0,0,0,0,0,0,0,0,0];
   pers string stGUISockPar{1}    := [""];
   pers num nGUISockRetPars{10}   := [0,0,0,0,0,0,0,0,0,0];
   pers string stGUISockRetPar{1} := [""];

endmodule

--- Backups/Robo_open_v2/RAPID/TASK0/SYSMOD/pntcmds.sys ---
module pntcmds(sysmodule)
   !
   ! (C) Copyright 2007 ABB
   !



   pers num nIntCommand          := 0;
   pers num nIntInParams{10}     := [0,0,0,0,0,0,0,0,0,0];
   pers string stIntInParams{1}  := [""];
   pers num nIntOutParams{10}    := [0,0,0,0,0,0,0,0,0,0];
   pers string stIntOutParams{1} := [""];



endmodule

--- Backups/Robo_open_v2/RAPID/TASK0/SYSMOD/syselog.sys ---
module syselog(sysmodule)

   !
   ! (C) Copyright 2005 ABB
   !
   const num PNT_ELOG_INFO    := 1;
   const num PNT_ELOG_WARNING := 2;
   const num PNT_ELOG_ERROR   := 3;

   proc PntElog(
      num elog_number,
      num type_err,
      \string Arg1,
      \string Arg2,
      \string Arg3,
      \string Arg4,
      \string Arg5)

      ! SysFun1. Undocumented hidden function.
      ! Scope: Used to write internal messages in common/process elog.
      ! This function shall NOT be used by our customers.
      ! Type_err :
      !           1 = Information
      !           2 = Warning
      !           3 = Error

      const num domain_no := 13;
      var string stArg1 := ERRSTR_UNUSED;
      var string stArg2 := ERRSTR_UNUSED;
      var string stArg3 := ERRSTR_UNUSED;
      var string stArg4 := ERRSTR_UNUSED;
      var string stArg5 := ERRSTR_UNUSED;


      if Present(Arg1) stArg1 := Arg1;
      if Present(Arg2) stArg2 := Arg2;
      if Present(Arg3) stArg3 := Arg3;
      if Present(Arg4) stArg4 := Arg4;
      if Present(Arg5) stArg5 := Arg5;

      SysFun1
         domain_no,
         elog_number,
         type_err ,
         stArg1,
         stArg2,
         stArg3,
         stArg4,
         stArg5;
   error
      Break; ! Unhandled error.
   endproc

endmodule

--- Backups/Robo_open_v2/RAPID/TASK0/SYSMOD/tpusocks.sys ---
module tpusocks(sysmodule)

   pers num nTPUSockCmdId    := 0;
   pers num nTPUSockClientId := 0;
   pers num nTPUSockSerNo    := 0;

   pers num nTPUSockPars{10}      := [0,0,0,0,0,0,0,0,0,0];
   pers string stTPUSockPar{1}    := [""];
   pers num nTPUSockRetPars{10}   := [0,0,0,0,0,0,0,0,0,0];
   pers string stTPUSockRetPar{1} := [""];

endmodule

--- Backups/Robo_open_v2/RAPID/TASK1/SYSMOD/bfdata.sys ---
module bfdata(sysmodule)



   const num BF_FLUID_CHANNEL := 1;
   const num BF_APPLICATORS := 1;
   const num BF_CHANNELS := 5;
   const num BF_MATERIALS := 100;

   pers bool bImmediateFactor := true; ! Indicate if also set immediately.
   pers bool bSkipBrushFactor; ! Set for each cycle as needed.

   pers num nCurrentFactor{BF_APPLICATORS, BF_CHANNELS} :=
     [[100,100,100,100,100]]; ! Current factors used for the current job.

   pers num nGlobalFactor{BF_APPLICATORS, BF_CHANNELS} :=
     [[100,100,100,100,100]];

   pers num nMaterialFactor{BF_MATERIALS, BF_APPLICATORS, BF_CHANNELS} :=
    [[[100,100,100,100,100]],
     [[100,100,100,100,100]],
     [[100,100,100,100,100]],
     [[100,100,100,100,100]],
     [[100,100,100,100,100]],
     [[100,100,100,100,100]],
     [[100,100,100,100,100]],
     [[100,100,100,100,100]],
     [[100,100,100,100,100]],
     [[100,100,100,100,100]],
     [[100,100,100,100,100]],
     [[100,100,100,100,100]],
     [[100,100,100,100,100]],
     [[100,100,100,100,100]],
     [[100,100,100,100,100]],
     [[100,100,100,100,100]],
     [[100,100,100,100,100]],
     [[100,100,100,100,100]],
     [[100,100,100,100,100]],
     [[100,100,100,100,100]],
     [[100,100,100,100,100]],
     [[100,100,100,100,100]],
     [[100,100,100,100,100]],
     [[100,100,100,100,100]],
     [[100,100,100,100,100]],
     [[100,100,100,100,100]],
     [[100,100,100,100,100]],
     [[100,100,100,100,100]],
     [[100,100,100,100,100]],
     [[100,100,100,100,100]],
     [[100,100,100,100,100]],
     [[100,100,100,100,100]],
     [[100,100,100,100,100]],
     [[100,100,100,100,100]],
     [[100,100,100,100,100]],
     [[100,100,100,100,100]],
     [[100,100,100,100,100]],
     [[100,100,100,100,100]],
     [[100,100,100,100,100]],
     [[100,100,100,100,100]],
     [[100,100,100,100,100]],
     [[100,100,100,100,100]],
     [[100,100,100,100,100]],
     [[100,100,100,100,100]],
     [[100,100,100,100,100]],
     [[100,100,100,100,100]],
     [[100,100,100,100,100]],
     [[100,100,100,100,100]],
     [[100,100,100,100,100]],
     [[100,100,100,100,100]],
     [[100,100,100,100,100]],
     [[100,100,100,100,100]],
     [[100,100,100,100,100]],
     [[100,100,100,100,100]],
     [[100,100,100,100,100]],
     [[100,100,100,100,100]],
     [[100,100,100,100,100]],
     [[100,100,100,100,100]],
     [[100,100,100,100,100]],
     [[100,100,100,100,100]],
     [[100,100,100,100,100]],
     [[100,100,100,100,100]],
     [[100,100,100,100,100]],
     [[100,100,100,100,100]],
     [[100,100,100,100,100]],
     [[100,100,100,100,100]],
     [[100,100,100,100,100]],
     [[100,100,100,100,100]],
     [[100,100,100,100,100]],
     [[100,100,100,100,100]],
     [[100,100,100,100,100]],
     [[100,100,100,100,100]],
     [[100,100,100,100,100]],
     [[100,100,100,100,100]],
     [[100,100,100,100,100]],
     [[100,100,100,100,100]],
     [[100,100,100,100,100]],
     [[100,100,100,100,100]],
     [[100,100,100,100,100]],
     [[100,100,100,100,100]],
     [[100,100,100,100,100]],
     [[100,100,100,100,100]],
     [[100,100,100,100,100]],
     [[100,100,100,100,100]],
     [[100,100,100,100,100]],
     [[100,100,100,100,100]],
     [[100,100,100,100,100]],
     [[100,100,100,100,100]],
     [[100,100,100,100,100]],
     [[100,100,100,100,100]],
     [[100,100,100,100,100]],
     [[100,100,100,100,100]],
     [[100,100,100,100,100]],
     [[100,100,100,100,100]],
     [[100,100,100,100,100]],
     [[100,100,100,100,100]],
     [[100,100,100,100,100]],
     [[100,100,100,100,100]],
     [[100,100,100,100,100]],
     [[100,100,100,100,100]]];



     ! Helper function to allow "late binding" setting of the value.
     proc ImmediateFactor(bool bValue)
        bImmediateFactor := bValue;
     endproc



     ! Calculate actual volume to be used with the factor applied.
     proc RetrFactorComp(inout num nVolume, num nMaterial, num nApp)
        nVolume := nVolume *
                  (nGlobalFactor{nApp, BF_FLUID_CHANNEL} / 100) *
                  (nMaterialFactor{nMaterial, nApp, BF_FLUID_CHANNEL} / 100);
     endproc



     ! Calculate real volume to store (100% factor) with the factor applied.
     ! Must use currently used factor for the job, in case it was changed while painting!
     proc StoreFactorComp(inout num nVolume, num nApp)
        nVolume := nVolume / (nCurrentFactor{nAPP, BF_FLUID_CHANNEL} / 100);
     endproc



endmodule

--- Backups/Robo_open_v2/RAPID/TASK1/SYSMOD/config.sys ---
module config(sysmodule)



   local const num MAX_OPTIONS := 20;
   local const num MAX_AREA := 5;

   pers string stOptionNames{MAX_AREA, MAX_OPTIONS};
   pers string stOptionValues{MAX_AREA, MAX_OPTIONS};
   pers string stAreaMapping{MAX_AREA};
   pers stringdig sdAreaFileTimes{MAX_AREA} := ["1710267316", "0", "0", "0", "0"];

   pers bool bConfigSemaphore;



   local func num nAreaMap(string stArea)
      for i from 1 to Dim(stAreaMapping, 1) do
         if stArea = stAreaMapping{i}
            return i;
      endfor
      return 0;
   endfunc



   local func bool bNewAreaMap(string stArea)
      for i from 1 to Dim(stAreaMapping, 1) do
         if stAreaMapping{i} = "" then
            stAreaMapping{i} := stArea;
            return true;
         endif
      endfor
      return false;
   endfunc



   func string stPntRapidOption(string stArea, string stOption)
      var bool bDoReRead;
      var string stFilePath;
      var string stValue := "";
      var stringdig sdFileTime;
      var bool bTimeOut;

      WaitUntil TestAndSet(bConfigSemaphore) \MaxTime := 5 \TimeFlag := bTimeOut;
      if bTimeOut then
         PntElog 4068, PNT_ELOG_ERROR \Arg1 := stArea \Arg2 := stOption;
         bConfigSemaphore := false; ! To get out of a deadlock situation.
         return "";
      endif

      stFilePath := HOME_ROOT + stArea + ".xml";

      if nAreaMap(stArea) = 0 then
         ! Area not used before, create new mapping.
         if IsFile(stFilePath) then
            if not bNewAreaMap(stArea) then
               PntElog 4055, PNT_ELOG_ERROR \Arg1 := stArea \Arg2 := stOption;
               bConfigSemaphore := false;
               return "";
            endif
         else
            PntElog 4056, PNT_ELOG_ERROR \Arg1 := stArea \Arg2 := stOption;
            bConfigSemaphore := false;
            return "";
         endif
         bDoReRead := true;
      else
         if FileTime(stFilePath \ModifyTime, \StrDig := sdFileTime) > 0 and
            StrDigCmp(sdAreaFileTimes{nAreaMap(stArea)}, LT, sdFileTime) then
            sdAreaFileTimes{nAreaMap(stArea)} := sdFileTime;
            bDoReRead := true;
         else
            bDoReRead := false;
         endif
      endif

      if bDoReRead then
         if nParseXMLFile(stFilePath, stOptionNames, stOptionValues, nAreaMap(stArea)) = 0 then
            PntElog 4057, PNT_ELOG_ERROR \Arg1 := stArea \Arg2 := stOption;
            bConfigSemaphore := false;
            return "";
         endif
      endif

      bConfigSemaphore := false;

      for i from 1 to Dim(stOptionNames, 2) do
         ! Case in-sensitive compare.
         if StrMap(stOptionNames{nAreaMap(stArea), i}, STR_LOWER, STR_UPPER) =
            StrMap(stArea + "/" + stOption, STR_LOWER, STR_UPPER)
            stValue := stOptionValues{nAreaMap(stArea), i};
      endfor

      if stValue = ""
         PntElog 4058, PNT_ELOG_ERROR \Arg1 := stArea \Arg2 := stOption;

      return stValue;
   error
      if errno = ERR_FILEACC then
         ! File has been deleted for some reason.
         PntElog 4062, PNT_ELOG_ERROR \Arg1 := stFilePath;
         bConfigSemaphore := false;
         return "";
      endif
   endfunc



   func bool bIsTrue(string stStatement)
      var num nTemp;

      ! Accept "1" as true.
      if StrToVal(stStatement, nTemp) then
         if nTemp = 1
            return true;
      endif

      ! Accept case insensitive "True" as true.
      if StrMap(stStatement, STR_LOWER, STR_UPPER) = "TRUE"
         return true;

      ! Accept case insensitive "Yes" as true.
      if StrMap(stStatement, STR_LOWER, STR_UPPER) = "YES"
         return true;

      return false;
   endfunc



   ! Very simple XML parser with only one stack depth (called the area).
   local func num nParseXMLFile(string stFileName, inout string stNames{*,*}, inout string stValues{*,*}, num nFirstDimension)
      var iodev ioFile;
      var string stLine;
      var string stCurrentArea := "";
      var num nOptionCount := 1;

      if nFirstDimension > Dim(stNames, 1) or nFirstDimension > Dim(stValues, 1) then
         PntElog 4059, PNT_ELOG_ERROR;
         return 0;
      endif

      ! Options are saved as paths like "Kernel/LogEnable" as the first dimension.

      Open stFileName, ioFile \Read;
      while stLine <> EOF do
         stLine := ReadStr(ioFile \RemoveCR);
         if stLine <> EOF then
            if StrMatch(stLine, 1, "<?") < StrLen(stLine) then
               ! Skip the XML header.
            elseif StrFind(stLine, 1, "=") < StrLen(stLine) then
               ! Line contains equal sign, so it must be an option=value tag.
               if stCurrentArea <> "" then
                  stNames{nFirstDimension, nOptionCount} := stCurrentArea + "/" + stStringBetween(stLine, "<", " ");
               else
                  stNames{nFirstDimension, nOptionCount} := stStringBetween(stLine, "<", " ");
               endif
               stValues{nFirstDimension, nOptionCount} := stStringBetween(stLine, """", """");
               Incr nOptionCount;
               if nOptionCount > Dim(stNames, 2) or nOptionCount > Dim(stValues, 2) then
                  PntElog 4061, PNT_ELOG_ERROR \Arg1 := stFileName \Arg2 := ValToStr(nOptionCount - 1);
                  Close ioFile;
                  return nOptionCount - 1;
               endif
            else
               ! No equal sign means it must be an "area" tag.
               if StrFind(stLine, 1, "/") < StrLen(stLine) then
                  ! Containing slash means the "area" is finished.
                  stCurrentArea := "";
               else
                  ! No slash means start of new "area".
                  stCurrentArea := stStringBetween(stLine, "<", ">");
               endif
            endif
         endif
      endwhile
      Close ioFile;

      return nOptionCount - 1;
   error
      if errno = ERR_FILEOPEN then
         PntElog 4062, PNT_ELOG_ERROR \Arg1 := stFileName;
         return 0;
      endif
   endfunc



   local func string stStringBetween(string stString, string stStart, string stEnd)
      var num nStartPos;
      var num nEndPos;

      nStartPos := StrMatch(stString, 1, stStart);
      if nStartPos > StrLen(stString) then
         PntElog 4063, PNT_ELOG_ERROR;
         return "";
      endif

      nEndPos := StrMatch(stString, nStartPos + 1, stEnd);
      if nEndPos > StrLen(stString) then
         PntElog 4063, PNT_ELOG_ERROR;
         return "";
      endif

      return StrPart(stString, nStartPos + 1, (nEndPos - nStartPos - 1));
   endfunc



endmodule

--- Backups/Robo_open_v2/RAPID/TASK1/SYSMOD/constant.sys ---
module constant(sysmodule)
   !
   ! (C) Copyright 2007 ABB
   !



   ! Command results:
   const num CMD_OK          := 0;
   const num CMD_FAILED      := -1;
   const num CMD_UNKNOWN     := -2;
   const num CMD_NOT_MASTER  := -3;
   const num CMD_TIMEOUT     := -4;
   const num CMD_INVALID_VAL := -5;
   const num CMD_ILL_SYSMODE := -6;
   const num CMD_RES_UNAVAIL := -7;

   ! Predefined modules and files:
   const num HOMEPOS_MODULE  := 10001;
   const num MCPOS_MODULE    := 10002;
   const string SEGMENT_NDX  := "segments.ndx";
   const string NONE_MODULE  := "none";

   ! Filesystem, directories and extensions:
   const string HOME_ROOT       := "HOME:/";
   const string SYSTEM_ROOT     := "INTERNAL:/pntrapid/";
   const string PROGRAM_DIR     := "programs/";
   const string LOG_DIR         := "logs/";
   const string PERS_CONFIG_DIR := "robdata/";
   const string CUST_MAIN_DIR   := "custmain/";
   const string CUST_PNT_DIR    := "custpnt/";
   const string CUST_MC_DIR     := "custmc/";
   const string MODULE_EXT      := ".mod";
   const string SYSMODULE_EXT   := ".sys";

   ! Misc:
   const num IGNORE_MC           := 0;
   const num UNDEFINED_IO_SIG    := -1000000;
   const string SYSTEM_PROC_NAME := "main";

   ! Limits:
   const num MAX_APPLICATORS := 4;

   ! Legacy (commvar.sys stuff For backward compability):
   const string stMedia         := "HOME:";
   const string ST_EMPTY_STRING := "";
   const string ST_PRG_EXT      := ".mod";
   const dionum tpLow           := 0;
   const dionum tpHigh          := 1;
   const dionum tpEdge          := 2;
   const num SYS_UNITIALIZED    := 0;
   const num SYS_DISABLED       := 1;
   const num SYS_STOPPED        := 2;
   const num SYS_READY          := 3;
   const num SYS_IN_PROG_STOP   := 4;
   const num SYS_IN_PROG_RUN    := 5;



endmodule

--- Backups/Robo_open_v2/RAPID/TASK1/SYSMOD/custmain.sys ---
module custmain(sysmodule)



   proc InitCustMain()
      !
      ! This will be executed during startmain/cancel...
      !
      Subscribe PRE_MAIN, "PreMainCustom";
      Subscribe POST_MAIN, "PostMainCustom";
   endproc



   proc PreMainCustom()
      !
      ! This will be executed before a paint program...
      !
   endproc



   proc PostMainCustom()
      !
      ! This will be executed after a paint program...
      !
   endproc



endmodule

--- Backups/Robo_open_v2/RAPID/TASK1/SYSMOD/cycinfo.sys ---
module cycinfo(sysmodule)



   record recCycReport
      string stTag;
      string stInfo;
      string stStart;
      num nDuration;
   endrecord



   local const num MAX_CR_ENTRIES := 15;

   pers recCycReport CurrCycReport{MAX_CR_ENTRIES};
   pers recCycReport LastCycReport{MAX_CR_ENTRIES};

   pers num nCREntriesUsed := 0;



   proc InitCycInfo()
      CycReportRotate; ! Also rotate on cancel.
   endproc



   proc CycReportRotate()
      if nCREntriesUsed > 0 then
         for i from 1 to nCREntriesUsed do
            LastCycReport{i} := CurrCycReport{i};
         endfor
      endif
      for i from (nCREntriesUsed + 1) to Dim(LastCycReport, 1) do
         LastCycReport{i} := ["", "", "", 0];
      endfor

      nCREntriesUsed := 0;
      for i from 1 to Dim(CurrCycReport, 1) do
         CurrCycReport{i} := ["", "", "", 0];
      endfor
   endproc



   local func string stPadToTwo(num nValue)
     if nValue < 10 then
        return "0" + ValToStr(nValue);
     else
        return ValToStr(nValue);
     endif
   endfunc



   local func string stNumToCFormat(num nSeconds)
      var num nMinutes;
      var num nHours;
      var num nMilli;

      nMilli := nSeconds;
      nSeconds := Trunc(nSeconds);
      nMilli := Trunc((nMilli - nSeconds) * 100);

      nHours := nSeconds div 3600;
      nSeconds := nSeconds - (nHours * 3600);
      nMinutes := nSeconds div 60;
      nSeconds := nSeconds - (nMinutes * 60);

      return "0000-00-00 " + stPadToTwo(nHours) + ":" + stPadToTwo(nMinutes) + ":" + stPadToTwo(nSeconds) + "." + stPadToTwo(nMilli);
   endfunc



   proc CycReportUpdate(string stTag \string stStart \string stInfo \num nDuration)
      var num nEntry := -1;

      if stTag = ""
         return;

      ! Does tag exist already?
      for i from 1 to Dim(CurrCycReport, 1) do
         if CurrCycReport{i}.stTag = stTag then
            nEntry := i;
         endif
      endfor

      if nEntry = -1 then
         ! Allocate new tag.
         Incr nCREntriesUsed;
         if nCREntriesUsed > Dim(CurrCycReport, 1) then
            Decr nCREntriesUsed;
            return;
         endif
         nEntry := nCREntriesUsed;
         CurrCycReport{nEntry}.stTag := stTag;
      endif

      if Present(stStart) then
         if RobOS() then
            CurrCycReport{nEntry}.stStart := stStart;
         else
            Set doUpdateVClock;
            WaitDO doUpdateVClock, 0;
            CurrCycReport{nEntry}.stStart := stNumToCFormat(nVirtualClock);
         endif
      endif
      if Present(stInfo)
         CurrCycReport{nEntry}.stInfo := stInfo;
      if Present(nDuration)
         CurrCycReport{nEntry}.nDuration := nDuration;
   endproc



endmodule

--- Backups/Robo_open_v2/RAPID/TASK1/SYSMOD/global.sys ---
module global(sysmodule)
   !
   ! (C) Copyright 2007 ABB
   !



   pers num nCurrProgIndex;
   pers num nCurrMtrlIndex;
   pers num nCurrJobOption;
   pers num nCurrMtrlOption1;
   pers num nCurrMtrlOption2;
   pers bool bCurrExpedited;
   pers num nCurrJobID;

   pers num nDirectProgIndex;
   pers num nDirectJobOption;
   pers bool bDirectExpedited;
   pers string stDirectModule;

   pers string stCurrModule;
   pers num nLastCycleTime;

   pers num nApplicators;

   pers num nRobotState;
   pers num nApplicatorState;
   pers num nProcessState;

   pers num nMasterID{4}; ! 4 = MASTER_CLIENTS constant from master.sys.

   pers num nPntCmdState;
   pers num nGuiSocketPort;
   pers num nVirtualClock;



endmodule

--- Backups/Robo_open_v2/RAPID/TASK1/SYSMOD/qextra.sys ---
module qextra(sysmodule)



   local const num EXTRA_COLUMNS := 3;

   ! Note: Size of the first dimension of this array
   ! have to correspond to the jobqueue size in qdata.sys.
   pers num nExtraQueue{10, EXTRA_COLUMNS} :=
      [[0,0,0],
       [0,0,0],
       [0,0,0],
       [0,0,0],
       [0,0,0],
       [0,0,0],
       [0,0,0],
       [0,0,0],
       [0,0,0],
       [0,0,0]];

   pers num nExtraBuffer{EXTRA_COLUMNS} :=
      [0,0,0];

   pers num nExtraCurrent{EXTRA_COLUMNS} :=
      [0,0,0];



endmodule

--- Backups/Robo_open_v2/RAPID/TASK1/SYSMOD/robdata.sys ---
module robdata(sysmodule)

   ! Note: This file can be used to add custom tools/speeds/zones.
   ! Uncomment any standard tools here, if they are needed.

   ! Robobel 925:
   pers tooldata tRB925_200 := [true,[[290.1,0,540],[0.866025,0,0.5,0]],[8,[0,0,33],[1,0,0,0],0,0,0]];
   pers tooldata tRB925_250 := [true,[[333.4,0,565],[0.866025,0,0.5,0]],[8,[0,0,33],[1,0,0,0],0,0,0]];

   ! HCEBELL:
   pers tooldata tHCEBELL_0   := [true,[[142.9,0,427.5],[0.866025,0,0.5,0]],[10,[0,-40,250],[1,0,0,0],0,0,0]];
   pers tooldata tHCEBELL_150 := [true,[[272.8,0,502.5],[0.866025,0,0.5,0]],[11,[0,40,250],[1,0,0,0],0,0,0]];
   pers tooldata tHCEBELL_200 := [true,[[316.1,0,527.5],[0.866025,0,0.5,0]],[11,[0,40,250],[1,0,0,0],0,0,0]];
   pers tooldata tHCEBELL_250 := [true,[[359.4,0,552.5],[0.866025,0,0.5,0]],[11,[0,40,250],[1,0,0,0],0,0,0]];
   pers tooldata tHCEBELL_300 := [true,[[402.7,0,577.5],[0.866025,0,0.5,0]],[11,[0,40,250],[1,0,0,0],0,0,0]];

   ! Default generic gun (10x5cm, 60 degree):
   pers tooldata tDefGun_Tip := [true,[[50,0,100],[0.866025,0,0.5,0]],[2,[0,0,50],[1,0,0,0],0,0,0]];
   pers tooldata tDefGun_100 := [true,[[136.6,0,150],[0.866025,0,0.5,0]],[2,[0,0,50],[1,0,0,0],0,0,0]];
   pers tooldata tDefGun_200 := [true,[[223.2,0,200],[0.866025,0,0.5,0]],[2,[0,0,50],[1,0,0,0],0,0,0]];

   ! ABB Ecco Gun:
   !pers tooldata tEccoGun_Tip := [true,[[1.8,0,156.6],[0.965926,0,0.258819,0]],[2,[0,0,120],[1,0,0,0],0,0,0]];
   !pers tooldata tEccoGun_200 := [true,[[101.8,0,329.8],[0.965926,0,0.258819,0]],[2,[0,0,120],[1,0,0,0],0,0,0]];
   !pers tooldata tEccoGun_250 := [true,[[126.8,0,373.1],[0.965926,0,0.258819,0]],[2,[0,0,120],[1,0,0,0],0,0,0]];
   !pers tooldata tEccoGun_300 := [true,[[151.8,0,416.4],[0.965926,0,0.258819,0]],[2,[0,0,120],[1,0,0,0],0,0,0]];

   ! G1Direct (short bracket):
   !pers tooldata tG1Direct_300 := [true,[[571.58,0,450],[0.866025,0,0.5,0]],[6.6,[135.2,0,174.1],[1,0,0,0],0,0,0]];
   !pers tooldata tG1Direct_250 := [true,[[528.28,0,425],[0.866025,0,0.5,0]],[6.6,[135.2,0,174.1],[1,0,0,0],0,0,0]];
   !pers tooldata tG1Direct_200 := [true,[[484.97,0,400],[0.866025,0,0.5,0]],[6.6,[135.2,0,174.1],[1,0,0,0],0,0,0]];

   ! G1_Long Braket:
   !pers tooldata tG1V3_200L := [true,[[487,0,502.3],[0.866025,0,0.5,0]],[8,[140.6,0,170],[1,0,0,0],0,0,0]];
   !pers tooldata tG1V3_250L := [true,[[524,0,528.9],[0.866025,0,0.5,0]],[8,[140.6,0,170],[1,0,0,0],0,0,0]];
   !pers tooldata tG1V3_300L := [true,[[549,0,571.6],[0.866025,0,0.5,0]],[8,[140.6,0,170],[1,0,0,0],0,0,0]];

   ! Cartrige Bell:
   !pers tooldata tCBS_0   := [true,[[121.25,0,415],[0.866025,0,0.5,0]],[5.5,[30,0,225],[1,0,0,0],0,0,0]];
   !pers tooldata tCBS_100 := [true,[[207.85,0,465],[0.866025,0,0.5,0]],[5.5,[30,0,225],[1,0,0,0],0,0,0]];
   !pers tooldata tCBS_200 := [true,[[294.45,0,515],[0.866025,0,0.5,0]],[5.5,[30,0,225],[1,0,0,0],0,0,0]];
   !pers tooldata tCBS_250 := [true,[[337.75,0,540],[0.866025,0,0.5,0]],[5.5,[30,0,225],[1,0,0,0],0,0,0]];
   !pers tooldata tCBS_300 := [true,[[381.05,0,565],[0.866025,0,0.5,0]],[5.5,[30,0,225],[1,0,0,0],0,0,0]];

   ! Robobel 926:
   !pers tooldata tRB926TD_0   := [true,[[116.9,0,470],[0.866025,0,0.5,0]],[5.5,[30,0,225],[1,0,0,0],0,0,0]];
   !pers tooldata tRB926TD_100 := [true,[[203.5,0,520],[0.866025,0,0.5,0]],[5.5,[30,0,225],[1,0,0,0],0,0,0]];
   !pers tooldata tRB926TD_120 := [true,[[220.8,0,530],[0.866025,0,0.5,0]],[5.5,[30,0,225],[1,0,0,0],0,0,0]];
   !pers tooldata tRB926TD_150 := [true,[[246.8,0,545],[0.866025,0,0.5,0]],[5.5,[30,0,225],[1,0,0,0],0,0,0]];
   !pers tooldata tRB926TD_200 := [true,[[290.1,0,570],[0.866025,0,0.5,0]],[5.5,[30,0,225],[1,0,0,0],0,0,0]];
   !pers tooldata tRB926TD_250 := [true,[[333.4,0,595],[0.866025,0,0.5,0]],[5.5,[30,0,225],[1,0,0,0],0,0,0]];
   !pers tooldata tRB926TD_300 := [true,[[376.7,0,620],[0.866025,0,0.5,0]],[5.5,[30,0,225],[1,0,0,0],0,0,0]];

   ! Robobel 625TD:
   !pers tooldata tRB625TD_0   := [true,[[116.9,0,420],[0.866025,0,0.5,0]],[5.1,[30,0,215],[1,0,0,0],0,0,0]];
   !pers tooldata tRB625TD_150 := [true,[[246.8,0,495],[0.866025,0,0.5,0]],[5.1,[30,0,215],[1,0,0,0],0,0,0]];
   !pers tooldata tRB625TD_200 := [true,[[290.1,0,520],[0.866025,0,0.5,0]],[5.1,[30,0,215],[1,0,0,0],0,0,0]];
   !pers tooldata tRB625TD_250 := [true,[[333.4,0,545],[0.866025,0,0.5,0]],[5.1,[30,0,215],[1,0,0,0],0,0,0]];
   !pers tooldata tRB625TD_300 := [true,[[376.7,0,570],[0.866025,0,0.5,0]],[5.1,[30,0,215],[1,0,0,0],0,0,0]];

   ! Robobel 951TD:
   !pers tooldata tRB951TD_0   := [true,[[116.9,0,470],[0.866025,0,0.5,0]],[6.3,[30,0,220],[1,0,0,0],0,0,0]];
   !pers tooldata tRB951TD_100 := [true,[[203.5,0,520],[0.866025,0,0.5,0]],[6.3,[30,0,220],[1,0,0,0],0,0,0]];
   !pers tooldata tRB951TD_120 := [true,[[220.8,0,530],[0.866025,0,0.5,0]],[6.3,[30,0,220],[1,0,0,0],0,0,0]];
   !pers tooldata tRB951TD_150 := [true,[[246.8,0,545],[0.866025,0,0.5,0]],[6.3,[30,0,220],[1,0,0,0],0,0,0]];
   !pers tooldata tRB951TD_200 := [true,[[290.1,0,570],[0.866025,0,0.5,0]],[6.3,[30,0,220],[1,0,0,0],0,0,0]];
   !pers tooldata tRB951TD_250 := [true,[[333.4,0,595],[0.866025,0,0.5,0]],[6.3,[30,0,220],[1,0,0,0],0,0,0]];
   !pers tooldata tRB951TD_300 := [true,[[376.7,0,620],[0.866025,0,0.5,0]],[6.3,[30,0,220],[1,0,0,0],0,0,0]];

   ! Robobel 951CBS /40pai/50pai/70pai:
   !pers tooldata tRB951CBS_0   := [true,[[121.25,0,415],[0.866025,0,0.5,0]],[6.3,[55,0,225],[1,0,0,0],0,0,0]];
   !pers tooldata tRB951CBS_100 := [true,[[207.85,0,465],[0.866025,0,0.5,0]],[6.3,[55,0,225],[1,0,0,0],0,0,0]];
   !pers tooldata tRB951CBS_120 := [true,[[225.17,0,475],[0.866025,0,0.5,0]],[6.3,[55,0,225],[1,0,0,0],0,0,0]];
   !pers tooldata tRB951CBS_150 := [true,[[251.15,0,490],[0.866025,0,0.5,0]],[6.3,[55,0,225],[1,0,0,0],0,0,0]];
   !pers tooldata tRB951CBS_200 := [true,[[294.45,0,515],[0.866025,0,0.5,0]],[6.3,[55,0,225],[1,0,0,0],0,0,0]];
   !pers tooldata tRB951CBS_250 := [true,[[337.75,0,540],[0.866025,0,0.5,0]],[6.3,[55,0,225],[1,0,0,0],0,0,0]];
   !pers tooldata tRB951CBS_300 := [true,[[381.05,0,565],[0.866025,0,0.5,0]],[6.3,[55,0,225],[1,0,0,0],0,0,0]];

   ! Interior Robobel951CBS /30pai:
   !pers tooldata tInteriorCBS_0   := [true,[[99.6,0,402.5],[0.866025,0,0.5,0]],[6.3,[30,0,220],[1,0,0,0],0,0,0]];
   !pers tooldata tInteriorCBS_100 := [true,[[186.2,0,452.5],[0.866025,0,0.5,0]],[6.3,[30,0,220],[1,0,0,0],0,0,0]];
   !pers tooldata tInteriorCBS_120 := [true,[[246.8,0,487.5],[0.866025,0,0.5,0]],[6.3,[30,0,220],[1,0,0,0],0,0,0]];
   !pers tooldata tInteriorCBS_150 := [true,[[272.8,0,502.5],[0.866025,0,0.5,0]],[6.3,[30,0,220],[1,0,0,0],0,0,0]];
   !pers tooldata tInteriorCBS_200 := [true,[[316.1,0,527.5],[0.866025,0,0.5,0]],[6.3,[30,0,220],[1,0,0,0],0,0,0]];
   !pers tooldata tInteriorCBS_250 := [true,[[359.4,0,552.5],[0.866025,0,0.5,0]],[6.3,[30,0,220],[1,0,0,0],0,0,0]];
   !pers tooldata tInteriorCBS_300 := [true,[[402.7,0,577.5],[0.866025,0,0.5,0]],[6.3,[30,0,220],[1,0,0,0],0,0,0]];

   ! Interior Robobel951 /30pai:
   !pers tooldata tInterior951_0   := [true,[[138.6,0,482.5],[0.866025,0,0.5,0]],[6.3,[30,0,220],[1,0,0,0],0,0,0]];
   !pers tooldata tInterior951_100 := [true,[[225.17,0,532.5],[0.866025,0,0.5,0]],[6.3,[30,0,220],[1,0,0,0],0,0,0]];
   !pers tooldata tInterior951_120 := [true,[[242.49,0,542.5],[0.866025,0,0.5,0]],[6.3,[30,0,220],[1,0,0,0],0,0,0]];
   !pers tooldata tInterior951_150 := [true,[[268.47,0,557.5],[0.866025,0,0.5,0]],[6.3,[30,0,220],[1,0,0,0],0,0,0]];
   !pers tooldata tInterior951_200 := [true,[[311.77,0,582.5],[0.866025,0,0.5,0]],[6.3,[30,0,220],[1,0,0,0],0,0,0]];
   !pers tooldata tInterior951_250 := [true,[[355.07,0,607.5],[0.866025,0,0.5,0]],[6.3,[30,0,220],[1,0,0,0],0,0,0]];
   !pers tooldata tInterior951_300 := [true,[[398.37,0,632.5],[0.866025,0,0.5,0]],[6.3,[30,0,220],[1,0,0,0],0,0,0]];

   ! RB-1000CBS /1C0341/500ccTank or RB-1000WSC /1C0356/700cc:
   !pers tooldata tRB1000WSC_0     := [true,[[121.25,0,450],[0.866025,0,0.5,0]],[10,[-52,0,270],[1,0,0,0],0,0,0]];
   !pers tooldata tRB1000WSC_100   := [true,[[207.85,0,500],[0.866025,0,0.5,0]],[10,[-52,0,270],[1,0,0,0],0,0,0]];
   !pers tooldata tRB1000WSC_150   := [true,[[251.15,0,525],[0.866025,0,0.5,0]],[10,[-52,0,270],[1,0,0,0],0,0,0]];
   !pers tooldata tRB1000WSC_200   := [true,[[294.45,0,550],[0.866025,0,0.5,0]],[10,[-52,0,270],[1,0,0,0],0,0,0]];
   !pers tooldata tRB1000WSC_250   := [true,[[337.75,0,575],[0.866025,0,0.5,0]],[10,[-52,0,270],[1,0,0,0],0,0,0]];
   !pers tooldata tRB1000WSC_300   := [true,[[381.05,0,600],[0.866025,0,0.5,0]],[10,[-52,0,270],[1,0,0,0],0,0,0]];
   !pers tooldata tRB1000WSC_teach := [true,[[-259.801,0,230],[0.866025,0,0.5,0]],[10,[-52,0,270],[1,0,0,0],0,0,0]];

   ! RB-1000SAD (Robobel Type):
   !pers tooldata tRB1000SAD_0   := [true,[[181.9,0,472.5],[0.866025,0,0.5,0]],[10,[31,0,260],[1,0,0,0],0,0,0]];
   !pers tooldata tRB1000SAD_100 := [true,[[268.5,0,522.5],[0.866025,0,0.5,0]],[10,[31,0,260],[1,0,0,0],0,0,0]];
   !pers tooldata tRB1000SAD_150 := [true,[[311.8,0,547.5],[0.866025,0,0.5,0]],[10,[31,0,260],[1,0,0,0],0,0,0]];
   !pers tooldata tRB1000SAD_200 := [true,[[355.1,0,572.5],[0.866025,0,0.5,0]],[10,[31,0,260],[1,0,0,0],0,0,0]];
   !pers tooldata tRB1000SAD_250 := [true,[[398.4,0,597.5],[0.866025,0,0.5,0]],[10,[31,0,260],[1,0,0,0],0,0,0]];
   !pers tooldata tRB1000SAD_300 := [true,[[441.7,0,622.5],[0.866025,0,0.5,0]],[10,[31,0,260],[1,0,0,0],0,0,0]];

   ! RB-1000SSD (Robobel Type):
   !PERS tooldata tRB1000SSD_0   := [true,[[181.9,0,472.5],[0.866025,0,0.5,0]],[10,[31,0,260],[1,0,0,0],0,0,0]];
   !PERS tooldata tRB1000SSD_100 := [true,[[268.5,0,522.5],[0.866025,0,0.5,0]],[10,[31,0,260],[1,0,0,0],0,0,0]];
   !PERS tooldata tRB1000SSD_150 := [true,[[311.8,0,547.5],[0.866025,0,0.5,0]],[10,[31,0,260],[1,0,0,0],0,0,0]];
   !PERS tooldata tRB1000SSD_200 := [true,[[355.1,0,572.5],[0.866025,0,0.5,0]],[10,[31,0,260],[1,0,0,0],0,0,0]];
   !PERS tooldata tRB1000SSD_250 := [true,[[398.4,0,597.5],[0.866025,0,0.5,0]],[10,[31,0,260],[1,0,0,0],0,0,0]];
   !PERS tooldata tRB1000SSD_300 := [true,[[441.7,0,622.5],[0.866025,0,0.5,0]],[10,[31,0,260],[1,0,0,0],0,0,0]];



   ! Speed data:
   const speeddata vPaint50   := [50,300,1000,50];
   const speeddata vPaint100  := [100,300,100,100];
   const speeddata vPaint150  := [150,300,150,150];
   const speeddata vPaint200  := [200,300,200,200];
   const speeddata vPaint250  := [250,300,250,250];
   const speeddata vPaint300  := [300,300,300,300];
   const speeddata vPaint350  := [350,300,350,350];
   const speeddata vPaint400  := [400,300,400,400];
   const speeddata vPaint450  := [450,300,450,450];
   const speeddata vPaint500  := [500,300,500,500];
   const speeddata vPaint550  := [550,300,1000,500];
   const speeddata vPaint600  := [600,300,1000,500];
   const speeddata vPaint650  := [650,300,1000,500];
   const speeddata vPaint700  := [700,300,1000,500];
   const speeddata vPaint750  := [750,300,1000,500];
   const speeddata vPaint800  := [800,300,1000,500];
   const speeddata vPaint850  := [850,300,1000,500];
   const speeddata vPaint900  := [900,300,1000,500];
   const speeddata vPaint950  := [950,300,1000,500];
   const speeddata vPaint1000 := [1000,300,1000,500];
   const speeddata vPaint1100 := [1100,300,1000,500];
   const speeddata vPaint1200 := [1200,300,1000,500];
   const speeddata vPaint1300 := [1300,300,1000,500];
   const speeddata vPaint1400 := [1400,300,1000,500];
   const speeddata vPaint1500 := [1500,300,1000,500];
   const speeddata vPaint1600 := [1600,300,1000,500];
   const speeddata vPaint1700 := [1700,300,1000,500];
   const speeddata vPaint1800 := [1800,300,1000,500];
   const speeddata vPaint1900 := [1900,300,1000,500];
   const speeddata vPaint2000 := [2000,300,1000,500];
   const speeddata vPaint2100 := [2100,300,1000,500];
   const speeddata vPaint2200 := [2200,300,1000,500];
   const speeddata vPaint2300 := [2300,300,1000,500];
   const speeddata vPaint2400 := [2400,300,1000,500];
   const speeddata vPaint2500 := [2500,300,1000,500];

   ! Speed data (High Flow Bell):
   const speeddata vHFB50   := [50,150,50,50];
   const speeddata vHFB100  := [100,150,100,100];
   const speeddata vHFB150  := [150,150,150,150];
   const speeddata vHFB200  := [200,150,200,200];
   const speeddata vHFB250  := [250,150,250,250];
   const speeddata vHFB300  := [300,150,300,300];
   const speeddata vHFB350  := [350,150,350,350];
   const speeddata vHFB400  := [400,150,400,400];
   const speeddata vHFB450  := [450,150,450,450];
   const speeddata vHFB500  := [500,150,500,500];
   const speeddata vHFB550  := [550,150,1000,500];
   const speeddata vHFB600  := [600,150,1000,500];
   const speeddata vHFB650  := [650,150,1000,500];
   const speeddata vHFB700  := [700,150,1000,500];
   const speeddata vHFB750  := [750,150,1000,500];
   const speeddata vHFB800  := [800,150,1000,500];
   const speeddata vHFB850  := [850,150,1000,500];
   const speeddata vHFB900  := [900,150,1000,500];
   const speeddata vHFB950  := [950,150,1000,500];
   const speeddata vHFB1000 := [1000,150,1000,500];
   const speeddata vHFB1100 := [1100,150,1000,500];
   const speeddata vHFB1200 := [1200,150,1000,500];
   const speeddata vHFB1300 := [1300,150,1000,500];
   const speeddata vHFB1400 := [1400,150,1000,500];
   const speeddata vHFB1500 := [1500,150,1000,500];
   const speeddata vHFB1600 := [1600,150,1000,500];
   const speeddata vHFB1700 := [1700,150,1000,500];
   const speeddata vHFB1800 := [1800,150,1000,500];
   const speeddata vHFB1900 := [1900,150,1000,500];
   const speeddata vHFB2000 := [2000,150,1000,500];
   const speeddata vHFB2100 := [2100,150,1000,500];
   const speeddata vHFB2200 := [2200,150,1000,500];
   const speeddata vHFB2300 := [2300,150,1000,500];
   const speeddata vHFB2400 := [2400,150,1000,500];
   const speeddata vHFB2500 := [2500,150,1000,500];



   ! Zone data:
   const zonedata zPaint1   := [false,1,1,1,0.15,1,0.15];
   const zonedata zPaint5   := [false,5,8,8,0.8,8,0.8];
   const zonedata zPaint10  := [false,10,15,15,1.5,15,1.5];
   const zonedata zPaint15  := [false,15,23,23,2.3,23,2.3];
   const zonedata zPaint20  := [false,20,30,30,3,30,3];
   const zonedata zPaint30  := [false,30,45,45,4.5,45,4.5];
   const zonedata zPaint40  := [false,40,60,60,6,60,6];
   const zonedata zPaint50  := [false,50,75,75,7.5,75,7.5];
   const zonedata zPaint60  := [false,60,90,90,9,90,9];
   const zonedata zPaint80  := [false,80,120,120,12,120,12];
   const zonedata zPaint100 := [false,100,150,150,15,150,15];
   const zonedata zPaint150 := [false,150,225,225,23,225,23];
   const zonedata zPaint200 := [false,200,300,300,30,300,30];
   const zonedata zPaint250 := [false,250,375,375,37.5,375,37.5];
   const zonedata zPaint300 := [false,300,450,450,45,450,45];



   proc ConfSettingsOff()
      ConfJ \Off;
      ConfL \Off;
   endproc



endmodule

--- Backups/Robo_open_v2/RAPID/TASK1/SYSMOD/sysdata.sys ---
module sysdata(sysmodule)

   ! Warning: Do not remove standard data from this module.

   pers robtarget pHomePos   := [[0,0,0],[9E+09,9E+09,9E+09,9E+09],[-1,-1,1,0],[9E+09,9E+09,9E+09,9E+09,9E+09,9E+09]];
   pers robtarget pMtrlChPos := [[0,0,0],[9E+09,9E+09,9E+09,9E+09],[-1,-1,1,0],[9E+09,9E+09,9E+09,9E+09,9E+09,9E+09]];
   pers robtarget pReadyPos  := [[0,0,0],[9E+09,9E+09,9E+09,9E+09],[-1,-1,1,0],[9E+09,9E+09,9E+09,9E+09,9E+09,9E+09]];
   pers robtarget pUserPos   := [[0,0,0],[9E+09,9E+09,9E+09,9E+09],[-1,-1,1,0],[9E+09,9E+09,9E+09,9E+09,9E+09,9E+09]];

   pers jointtarget jHomePos   := [[9E+09,9E+09,9E+09,9E+09,9E+09,9E+09],[9E+09,9E+09,9E+09,9E+09,9E+09,0]];
   pers jointtarget jMtrlChPos := [[9E+09,9E+09,9E+09,9E+09,9E+09,9E+09],[9E+09,9E+09,9E+09,9E+09,9E+09,0]];
   pers jointtarget jReadyPos  := [[9E+09,9E+09,9E+09,9E+09,9E+09,9E+09],[9E+09,9E+09,9E+09,9E+09,9E+09,0]];
   pers jointtarget jUserPos   := [[9E+09,9E+09,9E+09,9E+09,9E+09,9E+09],[9E+09,9E+09,9E+09,9E+09,9E+09,0]];

   pers tooldata tUserTool0 := [TRUE,[[0,0,0],[1,0,0,0]],[0.001,[0,0,0.001],[1,0,0,0],0,0,0]];

endmodule

--- Backups/Robo_open_v2/RAPID/TASK3/SYSMOD/custpnt.sys ---
module custpnt(sysmodule)



   proc InitCustPnt()
      !
      ! This will be executed during startup...
      !
      Subscribe TOGGLE_PATASK, "ToggleCustom";
   endproc



   proc ToggleCustom()
      !
      ! This will be executed on ProgramToggle or CommandToggle,
      ! depending on what IO interface is installed.
      !
      ! WARNING: Do not put time-consuming instructions here,
      ! since this is run in a trap, and will block the IO interface.
      !
   endproc



   proc Cmd1001(num nInparams{*}, string stInparams{*}, inout num nOutparams{*}, inout string stOutparams{*})
      !
      ! Insert RAPID code for command here...
      !
      nOutparams{1} := CMD_OK;
   error
      nOutparams{1} := CMD_FAILED;
      return;
   endproc



   proc Cmd1002(num nInparams{*}, string stInparams{*}, inout num nOutparams{*}, inout string stOutparams{*})
      !
      ! Insert RAPID code for command here...
      !
      nOutparams{1} := CMD_OK;
   error
      nOutparams{1} := CMD_FAILED;
      return;
   endproc



endmodule

--- Backups/Robo_open_v2/RAPID/TASK3/SYSMOD/qdata.sys ---
module qdata(sysmodule)



   pers num nJobQueueSize := 0; ! Actual number of entries/jobs.

   pers recJobInfo JobQueue{10} :=
      [[0,0,0,0,0,0,0,false],
       [0,0,0,0,0,0,0,false],
       [0,0,0,0,0,0,0,false],
       [0,0,0,0,0,0,0,false],
       [0,0,0,0,0,0,0,false],
       [0,0,0,0,0,0,0,false],
       [0,0,0,0,0,0,0,false],
       [0,0,0,0,0,0,0,false],
       [0,0,0,0,0,0,0,false],
       [0,0,0,0,0,0,0,false]];



endmodule

--- Backups/Robo_open_v2/HOME/programs/calpos.mod ---
module calpos

   ! SCOPE: Universal calibration/sync position program.

   proc mainCalPos()
      var jointtarget jLocalCalPos;

      ! Dummy instruction for SetPP.
      WaitTime 1;

      ! Set default values for all axis.
      jLocalCalPos := [[9E+09,9E+09,9E+09,9E+09,9E+09,9E+09],[9E+09,9E+09,9E+09,9E+09,9E+09,0]];

      jLocalCalPos.robax.rax_1 := nArmCalPos("rob1_1");
      jLocalCalPos.robax.rax_2 := nArmCalPos("rob1_2");
      jLocalCalPos.robax.rax_3 := nArmCalPos("rob1_3");
      jLocalCalPos.robax.rax_4 := nArmCalPos("rob1_4");
      jLocalCalPos.robax.rax_5 := nArmCalPos("rob1_5");
      jLocalCalPos.robax.rax_6 := nArmCalPos("rob1_6");

      if nRobSerialPart() = 5500 then
         ! IRB5500 has special values on axis 5 and 6, just set to 0 as stated in the manual.
         jLocalCalPos.robax.rax_5 := 0;
         jLocalCalPos.robax.rax_6 := 0;
      endif

      if stSingleJoint("AX7_1") <> "" then
         ! 7-axis robot.
         jLocalCalPos.extax.eax_a := nArmCalPos(stSingleJoint("AX7_1") \NoConversion);
      elseif nArmCalPos("obp_3") <> 9E+09 then
         ! 3-axis TurnTable.
         !IndReset OBP,2\RefNum:=0\Short;
         !IndReset OBP,3\RefNum:=0\Short;
         jLocalCalPos.extax.eax_a := nArmCalPos("obp_1");
         jLocalCalPos.extax.eax_b := nArmCalPos("obp_2");
         jLocalCalPos.extax.eax_c := nArmCalPos("obp_3");
      elseif nArmCalPos("obp_2") <> 9E+09 then
         ! 2-axis TurnTable.
         jLocalCalPos.extax.eax_a := nArmCalPos("obp_1");
         jLocalCalPos.extax.eax_b := nArmCalPos("obp_2");
      elseif nArmCalPos("obp_1") <> 9E+09 then
         ! 1-axis TurnTable.
         jLocalCalPos.extax.eax_a := nArmCalPos("obp_1");
      elseif nArmCalPos("track1") <> 9E+09 then
         ! IRB5350-02.
         jLocalCalPos.robax.rax_4 := 0;
         jLocalCalPos.robax.rax_5 := 0;
         jLocalCalPos.robax.rax_6 := 0;
         jLocalCalPos.extax.eax_a := nArmCalPos("track1" \NoConversion);
      else
         ! Attempt to get values for 8-axis robot.
         jLocalCalPos.extax.eax_a := nArmCalPos("rob1_7" \NoConversion);
         jLocalCalPos.extax.eax_b := nArmCalPos("rob1_8" \NoConversion);
      endif

      if stSingleJoint("H1AngleAxis") <> "" then
         ! Global CBS.
         jLocalCalPos.extax.eax_b := 0;
         jLocalCalPos.extax.eax_c := 0;
         jLocalCalPos.extax.eax_d := 0;
         jLocalCalPos.extax.eax_e := 0;
      endif

      MoveAbsJ jLocalCalPos,v100,fine,tool0;
      Stop;
   endproc

   local func num nArmCalPos(string stArm \switch NoConversion)
      var num nCalPos;
      ReadCfgData "/MOC/ARM/" + stArm, "cal_position", nCalPos;
      if Present(NoConversion) then
         return nCalPos;
      else
         return Round(nCalPos * (180 / 3.1415926) \Dec := 3);
      endif
   error
      if errno = ERR_CFG_NOTFND then
         SkipWarn;
         return 9E+09;
      endif
   endfunc

   local func string stSingleJoint(string stSingle)
      var string stJoint;
      ReadCfgData "/MOC/SINGLE/" + stSingle, "use_joint", stJoint;
      return stJoint;
   error
      if errno = ERR_CFG_NOTFND then
         SkipWarn;
         return "";
      endif
   endfunc

   local func num nRobSerialPart()
      var string stPart;
      var num nPart;
      ReadCfgData "/MOC/ROBOT_SERIAL_NUMBER/PID", "robot_serial_number_high_part", stPart;
      if StrToVal(StrPart(stPart, 1, StrFind(stPart, 1, "_") - 1), nPart) then
         return nPart;
      else
         return 9E+09;
      endif
   error
      SkipWarn;
      return 9E+09;
   endfunc

endmodule

--- Backups/Robo_open_v2/HOME/programs/m1.mod ---
MODULE M1

  PROC mainM1()
     WaitTime 10;
  ENDPROC
ENDMODULE

--- Backups/Robo_open_v2/HOME/programs/m10001.mod ---
module m10001

   ! SCOPE: Motion program for home position.

   proc mainm10001()
      if jHomePos.robax.rax_1 = 9E+09 then
         ErrWrite \W, "Home position not taught!", "";
      else
         MoveAbsJ jHomePos,v300,fine,tUserTool0;
      endif
   endproc

endmodule

--- Backups/Robo_open_v2/HOME/programs/m2.mod ---
MODULE M2

  PROC mainM2()
     WaitTime 10;
  ENDPROC
ENDMODULE

--- Backups/Robo_open_v2/HOME/programs/m3.mod ---
MODULE M3

  PROC mainM3()
     WaitTime 10;
  ENDPROC
ENDMODULE

--- Backups/Robot_ISEP_IRB140/SYSPAR/EIO.cfg ---
EIO:CFG_1.0:5:0::
#
EIO_BUS:

      -Name "Virtual1" -ConnectorID "SIM1"

      -Name "DeviceNet1" -BusType "DNET" -ConnectorID "PCI1"\
      -ConnectorLabel "First DeviceNet"
#
EIO_UNIT_TYPE:

      -Name "Virtual" -VendorName "ABB" -ProductName "Virtual unit"

      -Name "DN_GENERIC" -BusType "DNET" -DN_ExplicitMsgEnabled \
      -DN_C1OutputSize -1 -DN_C1InputSize -1

      -Name "d320" -BusType "DNET" -VendorName "ABB Robotics"\
      -ProductName "120 Vac Unit" -DN_VendorId 75 -DN_ProductCode 1\
      -DN_DeviceType 7 -DN_MajorRev 1 -DN_ExplicitMsgEnabled  -DN_C1Interval 50\
      -DN_C1OutputSize 2 -DN_C1InputSize 2

      -Name "d327A" -BusType "DNET" -VendorName "ABB Robotics"\
      -ProductName "Combi Unit" -DN_VendorId 75 -DN_ProductCode 2\
      -DN_DeviceType 100 -DN_MajorRev 5 -DN_ExplicitMsgEnabled  -DN_C1Type "COS"\
      -DN_C1OutputSize 6 -DN_C1InputSize 2

      -Name "d328A" -BusType "DNET" -VendorName "ABB Robotics"\
      -ProductName "24 VDC Unit" -DN_VendorId 75 -DN_ProductCode 3\
      -DN_DeviceType 7 -DN_ExplicitMsgEnabled  -DN_C1Type "COS"\
      -DN_C1OutputSize 2 -DN_C1InputSize 2

      -Name "d332A" -BusType "DNET" -VendorName "ABB Robotics"\
      -ProductName "Relay Unit" -DN_VendorId 75 -DN_ProductCode 5\
      -DN_DeviceType 7 -DN_MajorRev 2 -DN_ExplicitMsgEnabled  -DN_C1Type "COS"\
      -DN_C1OutputSize 2 -DN_C1InputSize 2

      -Name "d355A" -BusType "DNET" -VendorName "ABB Robotics"\
      -ProductName "Analog Unit" -DN_VendorId 75 -DN_ProductCode 10\
      -DN_DeviceType 100 -DN_MajorRev 1 -DN_ExplicitMsgEnabled \
      -DN_C1Interval 50 -DN_C1OutputSize 8 -DN_C1InputSize 8

      -Name "d651" -BusType "DNET" -VendorName "ABB Robotics"\
      -ProductName "Combi Unit" -DN_VendorId 75 -DN_ProductCode 25\
      -DN_DeviceType 100 -DN_ExplicitMsgEnabled  -DN_C1Type "COS"\
      -DN_C1OutputSize 5 -DN_C1InputSize 1

      -Name "d652" -BusType "DNET" -VendorName "ABB Robotics"\
      -ProductName "24 VDC Unit" -DN_VendorId 75 -DN_ProductCode 26\
      -DN_DeviceType 7 -DN_ExplicitMsgEnabled  -DN_C1Type "COS"\
      -DN_C1OutputSize 2 -DN_C1InputSize 2

      -Name "d653" -BusType "DNET" -VendorName "ABB Robotics"\
      -ProductName "Relay Unit" -DN_VendorId 75 -DN_ProductCode 27\
      -DN_DeviceType 7 -DN_ExplicitMsgEnabled  -DN_C1Type "COS"\
      -DN_C1OutputSize 1 -DN_C1InputSize 1

      -Name "DN_SLAVE" -BusType "DNET" -VendorName "ABB Robotics" -DN_VendorId 8\
      -DN_ProductCode 12 -DN_DeviceType 12 -DN_ExplicitMsgEnabled \
      -DN_C1Interval 50 -DN_C1OutputSize 8 -DN_C1InputSize 8

      -Name "DN_INTERNAL_SLAVE" -BusType "DNET" -VendorName "ABB Robotics"\
      -ProductName "Internal DeviceNet Slave" -InternalSlave  -DN_C1OutputSize 8\
      -DN_C1InputSize 8

      -Name "d350B" -BusType "DNET" -VendorName "ABB Robotics"\
      -ProductName "RIO Adapter" -DN_VendorId 75 -DN_ProductCode 6\
      -DN_DeviceType 7 -DN_MajorRev 2 -DN_ExplicitMsgEnabled  -DN_C1Type "COS"\
      -DN_C1OutputSize -1 -DN_C1InputSize -1

      -Name "DN_SLAVE_FA" -BusType "DNET" -VendorName "ABB Robotics"\
      -ProductName "DeviceNet Fieldbus Adapter Slave" -DN_VendorId 75\
      -DN_ProductCode 98 -DN_DeviceType 12 -DN_MajorRev 2 -DN_MinorRev 1\
      -DN_ExplicitMsgEnabled  -DN_C1Type "COS" -DN_C1OutputSize 8\
      -DN_C1InputSize 8

      -Name "d351A" -BusType "DNET" -VendorName "ABB Robotics"\
      -ProductName "IBS Adapter" -DN_VendorId 75 -DN_ProductCode 7\
      -DN_DeviceType 7 -DN_MajorRev 1 -DN_ExplicitMsgEnabled  -DN_C1Type "COS"\
      -DN_C1OutputSize -1 -DN_C1InputSize -1

      -Name "d352A" -BusType "DNET" -VendorName "ABB Robotics"\
      -ProductName "PBUS Adapter" -DN_VendorId 75 -DN_ProductCode 8\
      -DN_DeviceType 7 -DN_MajorRev 1 -DN_ExplicitMsgEnabled  -DN_C1Type "COS"\
      -DN_C1OutputSize -1 -DN_C1InputSize -1

      -Name "d352B" -BusType "DNET" -VendorName "ABB Robotics"\
      -ProductName "PBUS Adapter" -DN_VendorId 75 -DN_ProductCode 8\
      -DN_DeviceType 7 -DN_MajorRev 1 -DN_ExplicitMsgEnabled  -DN_C1Type "COS"\
      -DN_C1OutputSize -1 -DN_C1InputSize -1

      -Name "d378A" -BusType "DNET" -VendorName "ABB Robotics"\
      -ProductName "CCLink Adapter" -DN_VendorId 75 -DN_ProductCode 17\
      -DN_DeviceType 7 -DN_MajorRev 1 -DN_ExplicitMsgEnabled  -DN_C1Interval 50\
      -DN_C1OutputSize -1 -DN_C1InputSize -1
#
EIO_COMMAND_TYPE:

      -Name "LinkAddr" -UnitType "d350B" -DefValue "1" -OrderNr 1\
      -DN_Path "6,20 64 24 01 30 01,C6,1"

      -Name "DataRate" -UnitType "d350B" -DefValue "0" -OrderNr 2\
      -DN_Path "6,20 64 24 01 30 02,C6,1"

      -Name "StartQ" -UnitType "d350B" -DefValue "0" -OrderNr 3\
      -DN_Path "6,20 64 24 01 30 03,C6,1"

      -Name "RackSize" -UnitType "d350B" -DefValue "0" -OrderNr 4\
      -DN_Path "6,20 64 24 01 30 04,C6,1"

      -Name "LastRack" -UnitType "d350B" -DefValue "0" -OrderNr 5\
      -DN_Path "6,20 64 24 01 30 05,C1,1"

      -Name "D350Breset" -UnitType "d350B" -DefValue "0" -OrderNr 6\
      -DN_Path "4,20 01 24 01,C1,1" -DN_Service 5

      -Name "DataWidth" -UnitType "d351A" -DefValue "3" -OrderNr 1\
      -DN_Path "6,20 65 24 01 30 01,C6,1"

      -Name "D351Areset" -UnitType "d351A" -DefValue "0" -OrderNr 2\
      -DN_Path "4,20 01 24 01,C1,1" -DN_Service 5

      -Name "MasterInputSize" -UnitType "d352A" -DefValue "1" -OrderNr 1\
      -DN_Path "6,20 67 24 01 30 02,C6,1"

      -Name "MasterOutputSize" -UnitType "d352A" -DefValue "1" -OrderNr 2\
      -DN_Path "6,20 67 24 01 30 03,C6,1"

      -Name "StationAddress" -UnitType "d352A" -DefValue "126" -OrderNr 3\
      -DN_Path "6,20 67 24 01 30 04,C6,1"

      -Name "D352Areset" -UnitType "d352A" -DefValue "0" -OrderNr 4\
      -DN_Path "4,20 01 24 01,C1,1" -DN_Service 5

      -Name "MasterInputSize_B" -UnitType "d352B" -DefValue "1" -OrderNr 1\
      -DN_Path "6,20 67 24 01 30 02,C6,1"

      -Name "MasterOutputSize_B" -UnitType "d352B" -DefValue "1" -OrderNr 2\
      -DN_Path "6,20 67 24 01 30 03,C6,1"

